# B&R Automation Studio project Kesim
Automation Studio 6.7.0.187; technology packages: mappCockpit 6.7.0, mappMotion 6.7.2, mappServices 6.7.1, mappView 6.7.0, OpcUaCs 6.7.0

## Configuration Config1

CPU X20CP1685, AutomationRuntime 6.7.6, Build 11.3.0, Vc 6.5.0

### Task classes (Cpu.sw)
```
Cyclic#4:
  Kesim <- SourceCode.Kesim.prg
  CncCtrl <- SourceCode.CncCtrl.prg
Libraries: MpBase, runtime, AsZip, FileIO, aLibFile, AsBrStr, standard, astime, sys_lib, McBase, MpAxis, McAcpAx, McPathGen, McAcpTrak, McAxGroup, McAxis, McProgInt, MpRecipe, MpUserX, MpCnc, MpFile, MpPackML, MpAlarmX, CoTrace, MpServer, CMS_CT
```

### Hardware
```
8EI8X8HWT10.xxxx-1 : 8EI8X8HWT10.xxxx-1 v2.4.0.0 (NodeNumber=1)  [PLK1 -> X20CP1685.IF3 [Cable Type=PowerlinkCable, Length=10, Version=1.0.0.3]]
  DriveConfiguration/Encoder/EncoderX41:
    InterfaceType = EnDat
  DriveConfiguration/Encoder/EncoderX42:
    InterfaceType = EnDat
  DriveConfiguration/Encoder/EncoderX43:
    InterfaceType = EnDat
  DriveConfiguration/Channel[1]/RealAxis:
    AxisReference = gMpLink_AxisQX
  DriveConfiguration/Channel[1]/RealAxis/Homing:
    RestorePositionVariable = 
  DriveConfiguration/Channel[2]/RealAxis:
    AxisReference = gMpLink_AxisQY
  DriveConfiguration/Channel[2]/RealAxis/Homing:
    RestorePositionVariable = 
  DriveConfiguration/Channel[3]/RealAxis:
    AxisReference = gMpLink_AxisQC
  DriveConfiguration/Channel[3]/RealAxis/Homing:
    RestorePositionVariable = 
X20CP1685 : X20CP1685 v1.9.0.0
  Connector IF2:
    ActivateDevice = 1
    Mode = Manual
    InternetAddress = 192.168.5.10
    SubnetMask = 255.255.255.0
  ConfigurationID = Kesim_Config1
  Simulation = 1
  MotionLoggerSize = 2048000
  FileDevice1
  FileDeviceName1 = USER
  FileDevicePath1 = USER_PATH
```

### AxesGroup.axesgroup - X20CP1685/mappMotion/3AxesCNCXYC/AxesGroup.axesgroup
```
Element gMpLink_CncXYZ (Type=axesgroup)
  Type = PathGenAxesGroup
    PhysicalAxes:
      JointAxes:
        JointAxis[1]:
          Name = QX
          AxisRef = gMpLink_AxisQX
        JointAxis[2]:
          Name = QY
          AxisRef = gMpLink_AxisQY
        JointAxis[3]:
          Name = QZ
          AxisRef = gMpLink_AxisQC
    MechanicalSystem:
      MechSysRef = MechSys_3AxCNCXYZ
    AxesGroupFeatures:
      FeatureRef[1] = Feature_Programs
      FeatureRef[2] = Feature_Jogging
  Alarms = None
```

### CNCAxisCfg.axis - X20CP1685/mappMotion/3AxesCNCXYC/CNCAxisCfg.axis
```
Element gMpLink_AxisQX (Type=axis)
  BaseType = LinearBounded
  MovementLimits = Internal
    Position:
      LowerLimit = -25000.0
      UpperLimit = 25000.0
    Velocity:
      Velocity = 500000.0
    Acceleration:
      Acceleration = 500000.0
    Deceleration:
      Deceleration = 500000.0
  Alarms = None
Element gMpLink_AxisQY (Type=axis)
  BaseType = LinearBounded
  MovementLimits = Internal
    Position:
      LowerLimit = -25000.0
      UpperLimit = 25000.0
    Velocity:
      Velocity = 500000.0
    Acceleration:
      Acceleration = 500000.0
    Deceleration:
      Deceleration = 500000.0
  Alarms = None
Element gMpLink_AxisQC (Type=axis)
  BaseType = RotaryBounded
  MovementLimits = Internal
    Position:
      LowerLimit = -25000.0
      UpperLimit = 25000.0
    Velocity:
      Velocity = 500000.0
    Acceleration:
      Acceleration = 500000.0
    Deceleration:
      Deceleration = 500000.0
  Alarms = None
```

### GroupFeat.axesgroupfeature - X20CP1685/mappMotion/3AxesCNCXYC/GroupFeat.axesgroupfeature
```
Element Feature_Programs (Type=axesgroupfeature)
  Type = Program
    Location = User
      UserLocation[1]:
        FileDevice = DEV_CNC
Element Feature_Jogging (Type=axesgroupfeature)
  Type = Jogging
```

### MotionCfg.mappmotioncfg - X20CP1685/mappMotion/MotionCfg.mappmotioncfg
```
Element MappMotionConfiguration (Type=mappmotioncfg)
  SharedAlarms:
    Axis = MpAlarmX
    ACOPOSmultiAuxiliarySupplyModule = MpAlarmX
    ACOPOSmultiPowerSupplyModule = MpAlarmX
    AxesGroup = MpAlarmX
    Assembly = MpAlarmX
    Segment = MpAlarmX
    Sector = MpAlarmX
    Shuttle = MpAlarmX
    CamOperations = MpAlarmX
  Diagnostics:
    Snapshot = NotUsed
```

### AlmXCore.mpalarmxcore - X20CP1685/mappServices/AlarmX/AlmXCore.mpalarmxcore
```
Element gMpLink_AlarmXCore (Type=mpalarmxcore)
  mapp.Gen:
    Enable = TRUE
    EnableCockpit = TRUE
    TaskClass = 1
    Parent
  mapp.AlarmX.Core:
    Mapping:
      [0]:
        Alarm = [0]
        Action = Reaction
          Name = Category0_Abort
      [1]:
        Alarm = [1]
        Action = Reaction
          Name = Category1_Stop
      [2]:
        Alarm = [2]
        Action = Reaction
          Name = Category2_Pause
      [3]:
        Alarm = [3]
        Action = Reaction
          Name = Category3_Info
  mapp.AlarmX.List:
    [0]:
      List = gMpLink_AlarmXList_Abort
      Offset = 0
    [1]:
      List = gMpLink_AlarmXList_Stop
      Offset = 0
    [2]:
      List = gMpLink_AlarmXList_Info
      Offset = 0
  mapp.AlarmX.Create = Disabled
  mapp.AlarmX.Core.Retain:
    Memory = 0
  mapp.AlarmX.Core.Categories:
    [0]:
      List = gMpLink_AlarmXCategory
```

- AlmXLAbort.mpalarmxlist (1706109 bytes, not shown)

### RecipeXml.mprecipexml - X20CP1685/mappServices/Recipe/RecipeXml.mprecipexml
```
Element gMpLink_RecipeXml_Product (Type=mprecipexml)
  mapp.Gen:
    Enable = TRUE
    EnableCockpit = TRUE
    TaskClass = 4
    Audit = TRUE
    Parent
  mapp.Recipe.Xml:
    AutoSave = Standard
    Encryption = FALSE
    PassPhrase
    AutoExtension = TRUE
    Signature = Disabled
  Alarms = MpAlarmX
    mapp.AlarmX.Core.Configuration:
      [0]:
        Name = SaveFailed
        Message = {$BR/mapp/MpRecipeXml/Alarms/SaveFailed}
        Code = 0
        Severity = 1
        Behavior = EdgeAlarm
          AutoReset = TRUE
          Acknowledge = 1
          Confirm = 0
          MultipleInstances = TRUE
          ReactionWhilePending = TRUE
          Async = FALSE
          Recording:
            InactiveToActive = TRUE
            ActiveToInactive = FALSE
            UnacknowledgedToAcknowledged = TRUE
            UnconfirmedToConfirmed = TRUE
        Disable = FALSE
        AdditionalInformation1
        AdditionalInformation2
      [1]:
        Name = SaveFailedPartial
        Message = {$BR/mapp/MpRecipeXml/Alarms/SaveFailedPartial}
        Code = 0
        Severity = 1
        Behavior = EdgeAlarm
          AutoReset = TRUE
          Acknowledge = 1
          Confirm = 0
          MultipleInstances = TRUE
          ReactionWhilePending = TRUE
          Async = FALSE
          Recording:
            InactiveToActive = TRUE
            ActiveToInactive = FALSE
            UnacknowledgedToAcknowledged = TRUE
            UnconfirmedToConfirmed = TRUE
        Disable = FALSE
        AdditionalInformation1
        AdditionalInformation2
      [2]:
        Name = LoadFailed
        Message = {$BR/mapp/MpRecipeXml/Alarms/LoadFailed}
        Code = 0
        Severity = 1
        Behavior = EdgeAlarm
          AutoReset = TRUE
          Acknowledge = 1
          Confirm = 0
          MultipleInstances = TRUE
          ReactionWhilePending = TRUE
          Async = FALSE
          Recording:
            InactiveToActive = TRUE
            ActiveToInactive = FALSE
            UnacknowledgedToAcknowledged = TRUE
            UnconfirmedToConfirmed = TRUE
        Disable = FALSE
        AdditionalInformation1
        AdditionalInformation2
      [3]:
        Name = LoadFailedPartial
        Message = {$BR/mapp/MpRecipeXml/Alarms/LoadFailedPartial}
        Code = 0
        Severity = 1
        Behavior = EdgeAlarm
          AutoReset = TRUE
          Acknowledge = 1
          Confirm = 0
          MultipleInstances = TRUE
          ReactionWhilePending = TRUE
          Async = FALSE
          Recording:
            InactiveToActive = TRUE
            ActiveToInactive = FALSE
            UnacknowledgedToAcknowledged = TRUE
            UnconfirmedToConfirmed = TRUE
        Disable = FALSE
        AdditionalInformation1
        AdditionalInformation2
Element gMpLink_RecipeXml_Machine (Type=mprecipexml)
  mapp.Gen:
    Enable = TRUE
    EnableCockpit = TRUE
    TaskClass = 4
    Audit = TRUE
    Parent
  mapp.Recipe.Xml:
    AutoSave = Standard
    Encryption = FALSE
    PassPhrase
    AutoExtension = TRUE
    Signature = Disabled
  Alarms = MpAlarmX
    mapp.AlarmX.Core.Configuration:
      [0]:
        Name = SaveFailed
        Message = {$BR/mapp/MpRecipeXml/Alarms/SaveFailed}
        Code = 0
        Severity = 1
        Behavior = EdgeAlarm
          AutoReset = TRUE
          Acknowledge = 1
          Confirm = 0
          MultipleInstances = TRUE
          ReactionWhilePending = TRUE
          Async = FALSE
          Recording:
            InactiveToActive = TRUE
            ActiveToInactive = FALSE
            UnacknowledgedToAcknowledged = TRUE
            UnconfirmedToConfirmed = TRUE
        Disable = FALSE
        AdditionalInformation1
        AdditionalInformation2
      [1]:
        Name = SaveFailedPartial
        Message = {$BR/mapp/MpRecipeXml/Alarms/SaveFailedPartial}
        Code = 0
        Severity = 1
        Behavior = EdgeAlarm
          AutoReset = TRUE
          Acknowledge = 1
          Confirm = 0
          MultipleInstances = TRUE
          ReactionWhilePending = TRUE
          Async = FALSE
          Recording:
            InactiveToActive = TRUE
            ActiveToInactive = FALSE
            UnacknowledgedToAcknowledged = TRUE
            UnconfirmedToConfirmed = TRUE
        Disable = FALSE
        AdditionalInformation1
        AdditionalInformation2
      [2]:
        Name = LoadFailed
        Message = {$BR/mapp/MpRecipeXml/Alarms/LoadFailed}
        Code = 0
        Severity = 1
        Behavior = EdgeAlarm
          AutoReset = TRUE
          Acknowledge = 1
          Confirm = 0
          MultipleInstances = TRUE
          ReactionWhilePending = TRUE
          Async = FALSE
          Recording:
            InactiveToActive = TRUE
            ActiveToInactive = FALSE
            UnacknowledgedToAcknowledged = TRUE
            UnconfirmedToConfirmed = TRUE
        Disable = FALSE
        AdditionalInformation1
        AdditionalInformation2
      [3]:
        Name = LoadFailedPartial
        Message = {$BR/mapp/MpRecipeXml/Alarms/LoadFailedPartial}
        Code = 0
        Severity = 1
        Behavior = EdgeAlarm
          AutoReset = TRUE
          Acknowledge = 1
          Confirm = 0
          MultipleInstances = TRUE
          ReactionWhilePending = TRUE
          Async = FALSE
          Recording:
            InactiveToActive = TRUE
            ActiveToInactive = FALSE
            UnacknowledgedToAcknowledged = TRUE
            UnconfirmedToConfirmed = TRUE
        Disable = FALSE
        AdditionalInformation1
        AdditionalInformation2
```

### UsrX.mpuserx - X20CP1685/mappServices/UserX/UsrX.mpuserx
```
Element UserMgmtX (Type=mpuserx)
  mapp.Gen:
    Audit = TRUE
  UserMgmtSystem:
    UserMgmtSystemType = 0
  ServerSettings:
    Server = ADServer
      Timeout = 10
      Mapping:
        TableName
      DisplayName = Username
      AdditionalUserData:
        [0] = mail
        [1] = telephoneNumber
  PasswordPolicy:
    PasswordMaxAge = 0
    PasswordExpirationNotification = 0
    PasswordHistory = 0
    PasswordChangeReq = FALSE
    PasswordCase = FALSE
    PasswordAlpha = FALSE
    PasswordSpecial = FALSE
    PasswordLength = 2
  UserAccount:
    InvalidPasswordAttempts = 5
    UserExpirationTime = 0
    AutoLogoutTime = 3600
    UserNameLength = 1
    NoDelete = FALSE
    AdminUnlockTime = 0
    EditSameLevel = 1
  ImportExport:
    ImportUser = 2
    ImportRole = 2
    ImportUnchecked = FALSE
  Roles:
    DefRole#1:
      id = AdministratorBR
      level = 100
      admin = TRUE
    DefRole#2:
      id = AdministratorCU
      level = 90
      admin = TRUE
    DefRole#3:
      id = Supervisor
      level = 80
      admin = TRUE
    DefRole#4:
      id = Operator
      level = 70
      admin = TRUE
```

## Configuration FCL

CPU X20CP1685, AutomationRuntime 6.7.6, Build 11.3.0

### Hardware
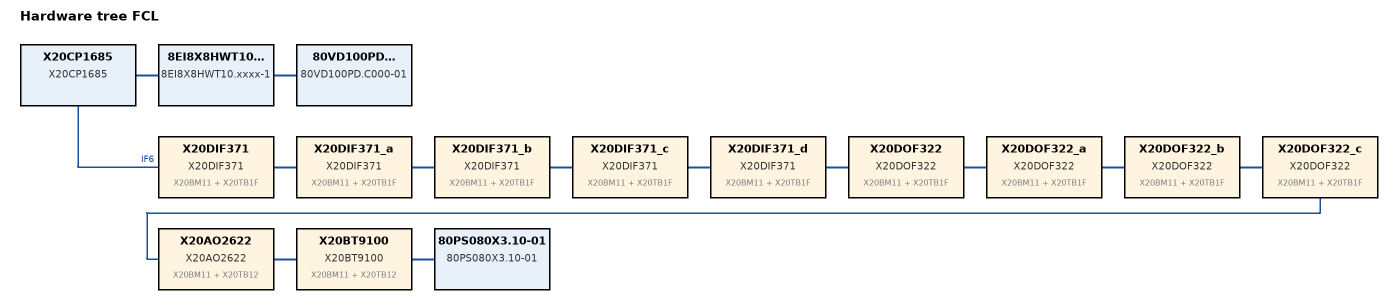
```
80PS080X3.10-01 : 80PS080X3.10-01 v1.7.0.0  [X2X1 -> X20BT9100.X2X1 [Cable Type=X2XCable, Length=10, Version=1.0.0.3]]
80VD100PD.C000-01 : 80VD100PD.C000-01 v2.5.1.0 (NodeNumber=2)  [PLK1 -> 8EI8X8HWT10.xxxx-1.PLK2 [Cable Type=PowerlinkCable, Length=10, Version=1.0.0.3]]
  EnableDNA = on
8EI8X8HWT10.xxxx-1 : 8EI8X8HWT10.xxxx-1 v2.4.0.0 (NodeNumber=1)  [PLK1 -> X20CP1685.IF3 [Cable Type=PowerlinkCable, Length=10, Version=1.0.0.3]; PLK2 -> 80VD100PD.C000-01.PLK1 [Cable Type=PowerlinkCable, Length=10, Version=1.0.0.3]]
  EnableDNA = on
X20AO2622 : X20AO2622 v1.5.0.0  [SS1 -> X20TB12.SS; SL -> X20BM11_i.SL1]
X20BM11 : X20BM11 v1.1.0.0  [X2X1 -> X20CP1685.IF6]
X20BM11_a : X20BM11 v1.1.0.0  [X2X1 -> X20BM11.X2X2]
X20BM11_b : X20BM11 v1.1.0.0  [X2X1 -> X20BM11_a.X2X2]
X20BM11_c : X20BM11 v1.1.0.0  [X2X1 -> X20BM11_b.X2X2]
X20BM11_d : X20BM11 v1.1.0.0  [X2X1 -> X20BM11_c.X2X2]
X20BM11_e : X20BM11 v1.1.0.0  [X2X1 -> X20BM11_d.X2X2]
X20BM11_f : X20BM11 v1.1.0.0  [X2X1 -> X20BM11_e.X2X2]
X20BM11_g : X20BM11 v1.1.0.0  [X2X1 -> X20BM11_f.X2X2]
X20BM11_h : X20BM11 v1.1.0.0  [X2X1 -> X20BM11_g.X2X2]
X20BM11_i : X20BM11 v1.1.0.0  [X2X1 -> X20BM11_h.X2X2]
X20BM11_j : X20BM11 v1.1.0.0  [X2X1 -> X20BM11_i.X2X2]
X20BT9100 : X20BT9100 v1.4.0.0  [SS1 -> X20TB12_a.SS; SL -> X20BM11_j.SL1]
X20CP1685 : X20CP1685 v1.9.0.0
  Connector IF2:
    ActivateDevice = 1
  ConfigurationID = Kesim_Config1
  Simulation = 1
  FileDevice1
  FileDeviceName1 = USER
  FileDevicePath1 = USER_PATH
X20DIF371 : X20DIF371 v1.4.1.0  [SS1 -> X20TB1F.SS; SL -> X20BM11.SL1]
X20DIF371_a : X20DIF371 v1.4.1.0  [SS1 -> X20TB1F_a.SS; SL -> X20BM11_a.SL1]
X20DIF371_b : X20DIF371 v1.4.1.0  [SS1 -> X20TB1F_b.SS; SL -> X20BM11_b.SL1]
X20DIF371_c : X20DIF371 v1.4.1.0  [SS1 -> X20TB1F_c.SS; SL -> X20BM11_c.SL1]
X20DIF371_d : X20DIF371 v1.4.1.0  [SS1 -> X20TB1F_d.SS; SL -> X20BM11_d.SL1]
X20DOF322 : X20DOF322 v1.5.2.0  [SS1 -> X20TB1F_e.SS; SL -> X20BM11_e.SL1]
X20DOF322_a : X20DOF322 v1.5.2.0  [SS1 -> X20TB1F_f.SS; SL -> X20BM11_f.SL1]
X20DOF322_b : X20DOF322 v1.5.2.0  [SS1 -> X20TB1F_g.SS; SL -> X20BM11_g.SL1]
X20DOF322_c : X20DOF322 v1.5.2.0  [SS1 -> X20TB1F_h.SS; SL -> X20BM11_h.SL1]
X20TB12 : X20TB12 v1.0.0.0
X20TB12_a : X20TB12 v1.0.0.0
X20TB1F : X20TB1F v1.0.0.0
X20TB1F_a : X20TB1F v1.0.0.0
X20TB1F_b : X20TB1F v1.0.0.0
X20TB1F_c : X20TB1F v1.0.0.0
X20TB1F_d : X20TB1F v1.0.0.0
X20TB1F_e : X20TB1F v1.0.0.0
X20TB1F_f : X20TB1F v1.0.0.0
X20TB1F_g : X20TB1F v1.0.0.0
X20TB1F_h : X20TB1F v1.0.0.0
```

## Configuration OCKM

### Hardware
```
X20CP1685 : X20CP1685 v1.9.0.0
  Connector IF2:
    ActivateDevice = 1
  ConfigurationID = Kesim_Config1
  Simulation = 1
  FileDevice1
  FileDeviceName1 = USER
  FileDevicePath1 = USER_PATH
```

## Configuration Office

CPU X20CP1685, AutomationRuntime 6.7.6, Build 11.3.0

### Task classes (Cpu.sw)
```
Cyclic#1:
  CncCtrl <- Source.CncCtrl.prg
Cyclic#4:
  AlarmX <- Source.Infastructure.AlarmX.prg
  UserXMgr <- Source.Infastructure.UserXMgr.prg
DataObjects: McAcpSys
NcDataObjects: McDriveLog
Binaries: TCLang, FWRules, mvLoader, TCData, udbdef, ArSvcReg, McAcpSim, McAcpDrv, McMechSys, iomap, asfw, Role, ashwd, sysconf, TC, BRRole, arconfig, User, ashwac, UaCsConfig, mCoWebSc, AxesGroup, SyncModule, CNCAxisCfg, MotionCfg, GroupFeat, Settings, SyncUnit, MechSystem, Hierarchy, mvConfig, AlmXCore, UsrX, AlmXHist, AlmXList, AlmXCateg, UsrXLogin, RecipeXml
Libraries: ArSsl, DataObj, UaCoal, AsHW, ArCert, ArUser, UaCoalPrv, AsETH, powerlnk, AsArProf, brsystem, AsMem, AsIO, AsEPL, operator, runtime, AsIecCon, astime, aLibFile, FileIO, AsBrStr, standard, sys_lib, AsZip, McBase, MpBase, MpAxis, McAcpAx, McPathGen, McAcpTrak, McAxGroup, McAxis, McProgInt, MpCnc, CoTrace, MpRecipe, MpUserX, MpFile, MpPackML, MpAlarmX, MpServer, CMS_CT
```

### Hardware
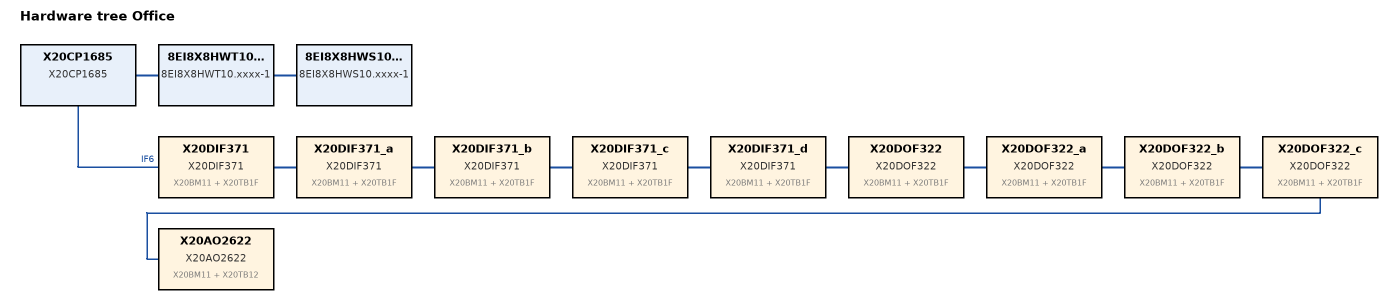
```
8EI8X8HWS10.xxxx-1 : 8EI8X8HWS10.xxxx-1 v2.4.0.0 (NodeNumber=2)  [PLK1 -> 8EI8X8HWT10.xxxx-1.PLK2 [Cable Type=PowerlinkCable, Length=10, Version=1.0.0.3]]
8EI8X8HWT10.xxxx-1 : 8EI8X8HWT10.xxxx-1 v2.4.0.0 (NodeNumber=1)  [PLK1 -> X20CP1685.IF3 [Cable Type=PowerlinkCable, Length=10, Version=1.0.0.3]; PLK2 -> 8EI8X8HWS10.xxxx-1.PLK1 [Cable Type=PowerlinkCable, Length=10, Version=1.0.0.3]]
  DriveConfiguration/Module:
    McAcoposTypeID = AcoposP3TConfig
    ActivateACOPOSSimulationOnPLC = 0
    PowerSupply = AC
  DriveConfiguration/Encoder/EncoderX41:
    InterfaceType = EnDat
  DriveConfiguration/Encoder/EncoderX42:
    InterfaceType = EnDat
  DriveConfiguration/Encoder/EncoderX43:
    InterfaceType = EnDat
  DriveConfiguration/Channel[1]/RealAxis:
    AxisReference = gMpLink_AxisQX
    MechanicalElementsIsInvisible = 0
  DriveConfiguration/Channel[1]/RealAxis/MechanicalElements/Gearbox:
    InputIsReadOnly = 0
    Input = 1
    OutputIsReadOnly = 0
    Output = 1
  DriveConfiguration/Channel[1]/RealAxis/MechanicalElements/RotaryToLinearTransformation:
    ReferenceDistanceIsReadOnly = 0
    ReferenceDistance = 1
  DriveConfiguration/Channel[1]/RealAxis:
    EncoderLink = OneEncoder
  DriveConfiguration/Channel[1]/RealAxis/Controller:
    ModeIsReadOnly = 0
    Mode = PositionController
  DriveConfiguration/Channel[1]/RealAxis/Homing:
    ModeIsReadOnly = 0
    Mode = Direct
    RestorePositionVariable = 
  DriveConfiguration/Channel[1]/RealAxis/StopReaction:
    QuickstopIsReadOnly = 0
    Quickstop = DecelerationLimit
    DriveErrorIsReadOnly = 0
    DriveError = DecelerationLimit
  DriveConfiguration/Channel[1]/RealAxis/MovementErrorLimits:
    PositionError = 10.0
    VelocityErrorMonitoring = Automatic1
  DriveConfiguration/Channel[1]/RealAxis:
    JerkFilterIsReadOnly = 0
    JerkFilter = NotUsed
    ZeroVibrationFilter = NotUsed
  DriveConfiguration/Channel[1]/RealAxis/DigitalInputs/HomingSwitch:
    SourceIsReadOnly = 0
    Source = NotUsed
    Level = High
  DriveConfiguration/Channel[1]/RealAxis/DigitalInputs/PositiveLimitSwitch:
    SourceIsReadOnly = 0
    Source = NotUsed
    Level = High
  DriveConfiguration/Channel[1]/RealAxis/DigitalInputs/NegativeLimitSwitch:
    SourceIsReadOnly = 0
    Source = NotUsed
    Level = High
  DriveConfiguration/Channel[1]/RealAxis/DigitalInputs/Trigger1:
    Source = X8Trigger1
    Level = High
  DriveConfiguration/Channel[1]/RealAxis/DigitalInputs/Trigger2:
    Source = X8Trigger2
    Level = High
  DriveConfiguration/Channel[1]/RealAxis/DigitalInputs/Quickstop:
    Input = Trigger2
  DriveConfiguration/Channel[1]/RealAxis/Simulation:
    SimulationModeOnPLC = SetValueGeneration
    SimulationModeOnACOPOS = NotUsed
  DriveConfiguration/Channel[1]:
    VirtualAxis = NotUsed
    ExternalEncoderAxis = NotUsed
  DriveConfiguration/Channel[2]/RealAxis:
    AxisReference = gMpLink_AxisQY
    MechanicalElementsIsInvisible = 0
  DriveConfiguration/Channel[2]/RealAxis/MechanicalElements/Gearbox:
    InputIsReadOnly = 0
    Input = 1
    OutputIsReadOnly = 0
    Output = 1
  DriveConfiguration/Channel[2]/RealAxis/MechanicalElements/RotaryToLinearTransformation:
    ReferenceDistanceIsReadOnly = 0
    ReferenceDistance = 1
  DriveConfiguration/Channel[2]/RealAxis:
    EncoderLink = OneEncoder
  DriveConfiguration/Channel[2]/RealAxis/Controller:
    ModeIsReadOnly = 0
    Mode = PositionController
  DriveConfiguration/Channel[2]/RealAxis/Homing:
    ModeIsReadOnly = 0
    Mode = Direct
    RestorePositionVariable = 
  DriveConfiguration/Channel[2]/RealAxis/StopReaction:
    QuickstopIsReadOnly = 0
    Quickstop = DecelerationLimit
    DriveErrorIsReadOnly = 0
    DriveError = DecelerationLimit
  DriveConfiguration/Channel[2]/RealAxis/MovementErrorLimits:
    PositionError = 10.0
    VelocityErrorMonitoring = Automatic1
  DriveConfiguration/Channel[2]/RealAxis:
    JerkFilterIsReadOnly = 0
    JerkFilter = NotUsed
    ZeroVibrationFilter = NotUsed
  DriveConfiguration/Channel[2]/RealAxis/DigitalInputs/HomingSwitch:
    SourceIsReadOnly = 0
    Source = NotUsed
    Level = High
  DriveConfiguration/Channel[2]/RealAxis/DigitalInputs/PositiveLimitSwitch:
    SourceIsReadOnly = 0
    Source = NotUsed
    Level = High
  DriveConfiguration/Channel[2]/RealAxis/DigitalInputs/NegativeLimitSwitch:
    SourceIsReadOnly = 0
    Source = NotUsed
    Level = High
  DriveConfiguration/Channel[2]/RealAxis/DigitalInputs/Trigger1:
    Source = X8Trigger1
    Level = High
  DriveConfiguration/Channel[2]/RealAxis/DigitalInputs/Trigger2:
    Source = X8Trigger2
    Level = High
  DriveConfiguration/Channel[2]/RealAxis/DigitalInputs/Quickstop:
    Input = Trigger2
  DriveConfiguration/Channel[2]/RealAxis/Simulation:
    SimulationModeOnPLC = SetValueGeneration
    SimulationModeOnACOPOS = NotUsed
  DriveConfiguration/Channel[2]:
    VirtualAxis = NotUsed
    ExternalEncoderAxis = NotUsed
  DriveConfiguration/Channel[3]/RealAxis:
    AxisReference = gMpLink_AxisQC
    MechanicalElementsIsInvisible = 0
  DriveConfiguration/Channel[3]/RealAxis/MechanicalElements/Gearbox:
    InputIsReadOnly = 0
    Input = 1
    OutputIsReadOnly = 0
    Output = 1
  DriveConfiguration/Channel[3]/RealAxis/MechanicalElements/RotaryToLinearTransformation:
    ReferenceDistanceIsReadOnly = 0
    ReferenceDistance = 1
  DriveConfiguration/Channel[3]/RealAxis:
    EncoderLink = OneEncoder
  DriveConfiguration/Channel[3]/RealAxis/Controller:
    ModeIsReadOnly = 0
    Mode = PositionController
  DriveConfiguration/Channel[3]/RealAxis/Homing:
    ModeIsReadOnly = 0
    Mode = Direct
    RestorePositionVariable = 
  DriveConfiguration/Channel[3]/RealAxis/StopReaction:
    QuickstopIsReadOnly = 0
    Quickstop = DecelerationLimit
    DriveErrorIsReadOnly = 0
    DriveError = DecelerationLimit
  DriveConfiguration/Channel[3]/RealAxis/MovementErrorLimits:
    PositionError = 10.0
    VelocityErrorMonitoring = Automatic1
  DriveConfiguration/Channel[3]/RealAxis:
    JerkFilterIsReadOnly = 0
    JerkFilter = NotUsed
    ZeroVibrationFilter = NotUsed
  DriveConfiguration/Channel[3]/RealAxis/DigitalInputs/HomingSwitch:
    SourceIsReadOnly = 0
    Source = NotUsed
    Level = High
  DriveConfiguration/Channel[3]/RealAxis/DigitalInputs/PositiveLimitSwitch:
    SourceIsReadOnly = 0
    Source = NotUsed
    Level = High
  DriveConfiguration/Channel[3]/RealAxis/DigitalInputs/NegativeLimitSwitch:
    SourceIsReadOnly = 0
    Source = NotUsed
    Level = High
  DriveConfiguration/Channel[3]/RealAxis/DigitalInputs/Trigger1:
    Source = X8Trigger1
    Level = High
  DriveConfiguration/Channel[3]/RealAxis/DigitalInputs/Trigger2:
    Source = X8Trigger2
    Level = High
  DriveConfiguration/Channel[3]/RealAxis/DigitalInputs/Quickstop:
    Input = Trigger2
  DriveConfiguration/Channel[3]/RealAxis/Simulation:
    SimulationModeOnPLC = SetValueGeneration
    SimulationModeOnACOPOS = NotUsed
  DriveConfiguration/Channel[3]:
    VirtualAxis = NotUsed
    ExternalEncoderAxis = NotUsed
X20AO2622 : X20AO2622 v1.5.0.0  [SS1 -> X20TB12.SS; SL -> X20BM11_i.SL1]
X20BM11 : X20BM11 v1.1.0.0  [X2X1 -> X20CP1685.IF6]
X20BM11_a : X20BM11 v1.1.0.0  [X2X1 -> X20BM11.X2X2]
X20BM11_b : X20BM11 v1.1.0.0  [X2X1 -> X20BM11_a.X2X2]
X20BM11_c : X20BM11 v1.1.0.0  [X2X1 -> X20BM11_b.X2X2]
X20BM11_d : X20BM11 v1.1.0.0  [X2X1 -> X20BM11_c.X2X2]
X20BM11_e : X20BM11 v1.1.0.0  [X2X1 -> X20BM11_d.X2X2]
X20BM11_f : X20BM11 v1.1.0.0  [X2X1 -> X20BM11_e.X2X2]
X20BM11_g : X20BM11 v1.1.0.0  [X2X1 -> X20BM11_f.X2X2]
X20BM11_h : X20BM11 v1.1.0.0  [X2X1 -> X20BM11_g.X2X2]
X20BM11_i : X20BM11 v1.1.0.0  [X2X1 -> X20BM11_h.X2X2]
X20CP1685 : X20CP1685 v1.9.0.0
  Connector IF2:
    ActivateDevice = 1
    ActivateSnmp = 2
  ConfigurationID = Cutting Table
  Simulation = 1
  MotionLoggerSize = 2048000
  EnableDebugger = 1
  TimerDeviceType = EPLX2X
  TimerDevice = X20CP1685.IF3
  TaskClassIdleTime = 2000
  Cyclic1Tolerance = 0
  FileDevice1
  FileDeviceName1 = USER
  FileDevicePath1 = USER_PATH
  ActivateFtpServer = 1
  ActivateWebServer = 1
  WebServerProtocol = 3
  ActivateSdm = 1
X20DIF371 : X20DIF371 v1.4.1.0  [SS1 -> X20TB1F.SS; SL -> X20BM11.SL1]
X20DIF371_a : X20DIF371 v1.4.1.0  [SS1 -> X20TB1F_a.SS; SL -> X20BM11_a.SL1]
X20DIF371_b : X20DIF371 v1.4.1.0  [SS1 -> X20TB1F_b.SS; SL -> X20BM11_b.SL1]
X20DIF371_c : X20DIF371 v1.4.1.0  [SS1 -> X20TB1F_c.SS; SL -> X20BM11_c.SL1]
X20DIF371_d : X20DIF371 v1.4.1.0  [SS1 -> X20TB1F_d.SS; SL -> X20BM11_d.SL1]
X20DOF322 : X20DOF322 v1.5.2.0  [SS1 -> X20TB1F_e.SS; SL -> X20BM11_e.SL1]
X20DOF322_a : X20DOF322 v1.5.2.0  [SS1 -> X20TB1F_f.SS; SL -> X20BM11_f.SL1]
X20DOF322_b : X20DOF322 v1.5.2.0  [SS1 -> X20TB1F_g.SS; SL -> X20BM11_g.SL1]
X20DOF322_c : X20DOF322 v1.5.2.0  [SS1 -> X20TB1F_h.SS; SL -> X20BM11_h.SL1]
X20TB12 : X20TB12 v1.0.0.0
X20TB1F : X20TB1F v1.0.0.0
X20TB1F_a : X20TB1F v1.0.0.0
X20TB1F_b : X20TB1F v1.0.0.0
X20TB1F_c : X20TB1F v1.0.0.0
X20TB1F_d : X20TB1F v1.0.0.0
X20TB1F_e : X20TB1F v1.0.0.0
X20TB1F_f : X20TB1F v1.0.0.0
X20TB1F_g : X20TB1F v1.0.0.0
X20TB1F_h : X20TB1F v1.0.0.0
```

### IoMap.iom - X20CP1685/IoMap.iom
```iecst
VAR_CONFIG
	::Kesim:fbCuttingTransfer_0.inEnable AT %IX."X20DIF371".DigitalInput01;
END_VAR
```

### PvMap.vvm - X20CP1685/PvMap.vvm
```iecst
VAR_CONFIG
	Cyclic#1.::ForceIO:slotIndex AT %Q.Cyclic#1.::gHMI.IO_Control.SelectedSlot; (*Insert your comment here...*)
	Cyclic#1.::ForceIO:GetSignalStr_0.eTypeSignal AT %Q.Cyclic#1.::gHMI.IO_Control.TypeOfIO; (*Insert your comment here...*)
END_VAR
```

### AxesGroup.axesgroup - X20CP1685/mappMotion/3AxesCNCXYC/AxesGroup.axesgroup
```
Element gMpLink_CncXYZ (Type=axesgroup)
  Type = PathGenAxesGroup
    PhysicalAxes:
      JointAxes:
        JointAxis[1]:
          Name = QX
          AxisRef = gMpLink_AxisQX
        JointAxis[2]:
          Name = QY
          AxisRef = gMpLink_AxisQY
        JointAxis[3]:
          Name = QC
          AxisRef = gMpLink_AxisQC
    MechanicalSystem:
      MechSysRef = MechSys_3AxCNCXYZ
    AxesGroupFeatures:
      FeatureRef[1] = Feature_Programs
      FeatureRef[2] = Feature_Jogging
```

### CNCAxisCfg.axis - X20CP1685/mappMotion/3AxesCNCXYC/CNCAxisCfg.axis
```
Element gMpLink_AxisQX (Type=axis)
  BaseType = LinearBounded
  MovementLimits = Internal
    Position:
      LowerLimit = -25000.0
      UpperLimit = 25000.0
    Velocity:
      Velocity = 500000.0
    Acceleration:
      Acceleration = 500000.0
    Deceleration:
      Deceleration = 500000.0
  Alarms = None
Element gMpLink_AxisQY (Type=axis)
  BaseType = LinearBounded
  MovementLimits = Internal
    Position:
      LowerLimit = -25000.0
      UpperLimit = 25000.0
    Velocity:
      Velocity = 500000.0
    Acceleration:
      Acceleration = 500000.0
    Deceleration:
      Deceleration = 500000.0
  Alarms = None
Element gMpLink_AxisQC (Type=axis)
  BaseType = RotaryBounded
  MovementLimits = Internal
    Position:
      LowerLimit = -25000.0
      UpperLimit = 25000.0
    Velocity:
      Velocity = 500000.0
    Acceleration:
      Acceleration = 500000.0
    Deceleration:
      Deceleration = 500000.0
  Alarms = None
```

### AxesGroup.axesgroup - X20CP1685/mappMotion/3AxesCNCXYZ/AxesGroup.axesgroup
```
Element gMpLink_CncXYZ (Type=axesgroup)
  Type = PathGenAxesGroup
    PhysicalAxes:
      JointAxes:
        JointAxis[1]:
          Name = QX
          AxisRef = gMpLink_AxisQX
        JointAxis[2]:
          Name = QY
          AxisRef = gMpLink_AxisQY
        JointAxis[3]:
          Name = VQZ
          AxisRef = gMpLink_AxisVQZ
    MechanicalSystem:
      MechSysRef = MechSys_3AxCNCXYZ
    AxesGroupFeatures:
      FeatureRef[1] = Feature_Programs
      FeatureRef[2] = Feature_Jogging
```

### CNCAxisCfg.axis - X20CP1685/mappMotion/3AxesCNCXYZ/CNCAxisCfg.axis
```
Element gMpLink_AxisQX (Type=axis)
  BaseType = LinearBounded
  MovementLimits:
    Position:
      LowerLimit = -25000.0
      UpperLimit = 25000.0
    Velocity:
      Velocity = 500000.0
    Acceleration:
      Acceleration = 500000.0
    Deceleration:
      Deceleration = 500000.0
Element gMpLink_AxisQY (Type=axis)
  BaseType = LinearBounded
  MovementLimits:
    Position:
      LowerLimit = -25000.0
      UpperLimit = 25000.0
    Velocity:
      Velocity = 500000.0
    Acceleration:
      Acceleration = 500000.0
    Deceleration:
      Deceleration = 500000.0
Element gMpLink_AxisVQZ (Type=axis)
  BaseType = LinearBounded
  MovementLimits:
    Position:
      LowerLimit = -25000.0
      UpperLimit = 25000.0
    Velocity:
      Velocity = 500000.0
    Acceleration:
      Acceleration = 500000.0
    Deceleration:
      Deceleration = 500000.0
Element gMpLink_AxisB (Type=axis)
  BaseType = RotaryBounded
  MovementLimits:
    Position:
      LowerLimit = -25000.0
      UpperLimit = 25000.0
    Velocity:
      Velocity = 500000.0
    Acceleration:
      Acceleration = 500000.0
    Deceleration:
      Deceleration = 500000.0
Element gMpLink_AxisC (Type=axis)
  BaseType = RotaryBounded
  MovementLimits:
    Position:
      LowerLimit = -25000.0
      UpperLimit = 25000.0
    Velocity:
      Velocity = 500000.0
    Acceleration:
      Acceleration = 500000.0
    Deceleration:
      Deceleration = 500000.0
```

### MechSystem.mechanicalsystem - X20CP1685/mappMotion/3AxesCNCXYZ/MechSystem.mechanicalsystem
```
Element MechSys_3AxCNCXYZ (Type=mechanicalsystem)
  Type = 3AxesCNC
    Subtype:
      JointAxesPositionLimits:
        JointAxis[1]
        JointAxis[2]
        JointAxis[3]
```

### MotionCfg.mappmotioncfg - X20CP1685/mappMotion/MotionCfg.mappmotioncfg
```
Element MappMotionConfiguration (Type=mappmotioncfg)
  Processing:
    ProcessingTaskClass = 1
    ExplicitComputationOrder:
      Axis = NotUsed
  Logger:
    SelectiveLogging = NotUsed
  SharedAlarms:
    Axis = MpAlarmX
    ACOPOSmultiAuxiliarySupplyModule = MpAlarmX
    ACOPOSmultiPowerSupplyModule = MpAlarmX
    AxesGroup = MpAlarmX
    Assembly = MpAlarmX
    Segment = MpAlarmX
    Sector = MpAlarmX
    Shuttle = MpAlarmX
    CamOperations = MpAlarmX
  McAcpDrv:
    POWERLINKCyclesPerParID = 2
```

### Config_3.purevaxcfg - X20CP1685/mappMotion/PureVAxis/Config_3.purevaxcfg
```
Element PureVAxCfg_1 (Type=purevaxcfg)
  PureVAxis:
    AxisReference = gMpLink_AxisVQZ
```

### AlmXCateg.mpalarmxcategory - X20CP1685/mappServices/AlarmX/AlmXCateg.mpalarmxcategory
```
Element gMpLink_AlarmXCategory (Type=mpalarmxcategory)
  mapp.AlarmX.Categories:
    [0]:
      Name = Category0_Abort
      SourceProperty = Severity
        Severity = 0
    [1]:
      Name = Category1_Stop
      SourceProperty = Severity
        Severity = 1
    [2]:
      Name = Category2_Pause
      SourceProperty = Severity
        Severity = 2
    [3]:
      Name = Category3_Info
      SourceProperty = Severity
        Severity = 3
```

### AlmXHist.mpalarmxhistory - X20CP1685/mappServices/AlarmX/AlmXHist.mpalarmxhistory
```
Element gMpLink_AlarmXHistory (Type=mpalarmxhistory)
  mapp.Gen:
    Enable = TRUE
    EnableCockpit = TRUE
    Audit = TRUE
    Parent
  mapp.AlarmX.History:
    Export:
      TimeStampPattern = %Y-%m-%d %H:%M:%S:%L
      AutoExtension = TRUE
      ColumnSeparator = ,
    Memory = 0
      Size = 2048
      BufferSize = 10
      Interval = 60
    Scope = 0
```

### AlmXLInfo.mpalarmxlist - X20CP1685/mappServices/AlarmX/AlmXLInfo.mpalarmxlist
```
Element gMpLink_AlarmXList_Info (Type=mpalarmxlist)
  mapp.AlarmX.Core.Configuration:
    [0]:
      Name = Alert.0
      Message = {&TextSnippet.0}{$AlarmX/Alerts/Alert.0}
      Code = 0
      Severity = 3
      Behavior = DiscreteValueMonitoring
        Confirm = 0
        ReactionWhilePending = TRUE
        Recording:
          InactiveToActive = TRUE
          UnacknowledgedToAcknowledged = TRUE
          AcknowledgedToUnacknowledged = FALSE
          UnconfirmedToConfirmed = TRUE
          ConfirmedToUnconfirmed = FALSE
          Update = FALSE
        Monitoring:
          MonitoredPV = ::AlarmX:Loc.Status.Alerts.Single.Info[0]
          TriggerValues:
            [0] = 1
          Settings = 0
            Delay = 0.0
      Disable = FALSE
      InhibitPV
      AdditionalInformation1
      AdditionalInformation2
    [1]:
      Name = Alert.1
      Message = {&TextSnippet.1}{$AlarmX/Alerts/Alert.1}
      Code = 1
      Severity = 2
      Behavior = DiscreteValueMonitoring
        Confirm = 0
        ReactionWhilePending = TRUE
        Recording:
          InactiveToActive = TRUE
          UnacknowledgedToAcknowledged = TRUE
          AcknowledgedToUnacknowledged = FALSE
          UnconfirmedToConfirmed = TRUE
          ConfirmedToUnconfirmed = FALSE
          Update = FALSE
        Monitoring:
          MonitoredPV = ::AlarmX:Loc.Status.Alerts.Single.Stop[1]
          TriggerValues:
            [0] = 1
          Settings = 0
            Delay = 0.0
      Disable = FALSE
      InhibitPV
      AdditionalInformation1
      AdditionalInformation2
    [2]:
      Name = Alert.2
      Message = {&TextSnippet.2}{$AlarmX/Alerts/Alert.2}
      Code = 2
      Severity = 2
      Behavior = DiscreteValueMonitoring
        Confirm = 0
        ReactionWhilePending = TRUE
        Recording:
          InactiveToActive = TRUE
          UnacknowledgedToAcknowledged = TRUE
          AcknowledgedToUnacknowledged = FALSE
          UnconfirmedToConfirmed = TRUE
          ConfirmedToUnconfirmed = FALSE
          Update = FALSE
        Monitoring:
          MonitoredPV = ::AlarmX:Loc.Status.Alerts.Single.Stop[2]
          TriggerValues:
            [0] = 1
          Settings = 0
            Delay = 0.0
      Disable = FALSE
      InhibitPV
      AdditionalInformation1
      AdditionalInformation2
    [3]:
      Name = Alert.3
      Message = {&TextSnippet.3}{$AlarmX/Alerts/Alert.3}
      Code = 3
      Severity = 2
      Behavior = DiscreteValueMonitoring
        Confirm = 0
        ReactionWhilePending = TRUE
        Recording:
          InactiveToActive = TRUE
          UnacknowledgedToAcknowledged = TRUE
          AcknowledgedToUnacknowledged = FALSE
          UnconfirmedToConfirmed = TRUE
          ConfirmedToUnconfirmed = FALSE
          Update = FALSE
        Monitoring:
          MonitoredPV = ::AlarmX:Loc.Status.Alerts.Single.Stop[3]
          TriggerValues:
            [0] = 1
          Settings = 0
            Delay = 0.0
      Disable = FALSE
      InhibitPV
      AdditionalInformation1
      AdditionalInformation2
    [4]:
      Name = Alert.4
      Message = {&TextSnippet.4}{$AlarmX/Alerts/Alert.4}
      Code = 4
      Severity = 2
      Behavior = DiscreteValueMonitoring
        Confirm = 0
        ReactionWhilePending = TRUE
        Recording:
          InactiveToActive = TRUE
          UnacknowledgedToAcknowledged = TRUE
          AcknowledgedToUnacknowledged = FALSE
          UnconfirmedToConfirmed = TRUE
          ConfirmedToUnconfirmed = FALSE
          Update = FALSE
        Monitoring:
          MonitoredPV = ::AlarmX:Loc.Status.Alerts.Single.Stop[4]
          TriggerValues:
            [0] = 1
          Settings = 0
            Delay = 0.0
      Disable = FALSE
      InhibitPV
      AdditionalInformation1
      AdditionalInformation2
    [5]:
      Name = Alert.5
      Message = {$AlarmX/Alerts/Alert.5}
      Code = 5
      Severity = 2
      Behavior = DiscreteValueMonitoring
        Confirm = 0
        ReactionWhilePending = TRUE
        Recording:
          InactiveToActive = TRUE
          UnacknowledgedToAcknowledged = TRUE
          AcknowledgedToUnacknowledged = FALSE
          UnconfirmedToConfirmed = TRUE
          ConfirmedToUnconfirmed = FALSE
          Update = FALSE
        Monitoring:
          MonitoredPV = ::AlarmX:Loc.Status.Alerts.Single.Stop[5]
          TriggerValues:
            [0] = 1
          Settings = 0
            Delay = 0.0
      Disable = FALSE
      InhibitPV
      AdditionalInformation1
      AdditionalInformation2
    [6]:
      Name = Alert.6
      Message = {$AlarmX/Alerts/Alert.6}
      Code = 6
      Severity = 2
      Behavior = DiscreteValueMonitoring
        Confirm = 0
        ReactionWhilePending = TRUE
        Recording:
          InactiveToActive = TRUE
          UnacknowledgedToAcknowledged = TRUE
          AcknowledgedToUnacknowledged = FALSE
          UnconfirmedToConfirmed = TRUE
          ConfirmedToUnconfirmed = FALSE
          Update = FALSE
        Monitoring:
          MonitoredPV = ::AlarmX:Loc.Status.Alerts.Single.Stop[6]
          TriggerValues:
            [0] = 1
          Settings = 0
            Delay = 0.0
      Disable = FALSE
      InhibitPV
      AdditionalInformation1
      AdditionalInformation2
    [7]:
      Name = Alert.7
      Message = {$AlarmX/Alerts/Alert.7}
      Code = 7
      Severity = 2
      Behavior = DiscreteValueMonitoring
        Confirm = 0
        ReactionWhilePending = TRUE
        Recording:
          InactiveToActive = TRUE
          UnacknowledgedToAcknowledged = TRUE
          AcknowledgedToUnacknowledged = FALSE
          UnconfirmedToConfirmed = TRUE
          ConfirmedToUnconfirmed = FALSE
          Update = FALSE
        Monitoring:
          MonitoredPV = ::AlarmX:Loc.Status.Alerts.Single.Stop[7]
          TriggerValues:
            [0] = 1
          Settings = 0
            Delay = 0.0
      Disable = FALSE
      InhibitPV
      AdditionalInformation1
      AdditionalInformation2
    [8]:
      Name = Alert.8
      Message = {$AlarmX/Alerts/Alert.8}
      Code = 8
      Severity = 2
      Behavior = DiscreteValueMonitoring
        Confirm = 0
        ReactionWhilePending = TRUE
        Recording:
          InactiveToActive = TRUE
          UnacknowledgedToAcknowledged = TRUE
          AcknowledgedToUnacknowledged = FALSE
          UnconfirmedToConfirmed = TRUE
          ConfirmedToUnconfirmed = FALSE
          Update = FALSE
        Monitoring:
          MonitoredPV = ::AlarmX:Loc.Status.Alerts.Single.Stop[8]
          TriggerValues:
            [0] = 1
          Settings = 0
            Delay = 0.0
      Disable = FALSE
      InhibitPV
      AdditionalInformation1
      AdditionalInformation2
    [9]:
      Name = Alert.9
      Message = {$AlarmX/Alerts/Alert.9}
      Code = 9
      Severity = 2
      Behavior = DiscreteValueMonitoring
        Confirm = 0
        ReactionWhilePending = TRUE
        Recording:
          InactiveToActive = TRUE
          UnacknowledgedToAcknowledged = TRUE
          AcknowledgedToUnacknowledged = FALSE
          UnconfirmedToConfirmed = TRUE
          ConfirmedToUnconfirmed = FALSE
          Update = FALSE
        Monitoring:
          MonitoredPV = ::AlarmX:Loc.Status.Alerts.Single.Stop[9]
          TriggerValues:
            [0] = 1
          Settings = 0
            Delay = 0.0
      Disable = FALSE
      InhibitPV
      AdditionalInformation1
      AdditionalInformation2
    [10]:
      Name = Alert.10
      Message = {$AlarmX/Alerts/Alert.10}
      Code = 10
      Severity = 2
      Behavior = DiscreteValueMonitoring
        Confirm = 0
        ReactionWhilePending = TRUE
        Recording:
          InactiveToActive = TRUE
          UnacknowledgedToAcknowledged = TRUE
          AcknowledgedToUnacknowledged = FALSE
          UnconfirmedToConfirmed = TRUE
          ConfirmedToUnconfirmed = FALSE
          Update = FALSE
        Monitoring:
          MonitoredPV = ::AlarmX:Loc.Status.Alerts.Single.Stop[10]
          TriggerValues:
            [0] = 1
          Settings = 0
            Delay = 0.0
      Disable = FALSE
      InhibitPV
      AdditionalInformation1
      AdditionalInformation2
    [11]:
      Name = Alert.11
      Message = {$AlarmX/Alerts/Alert.11}
      Code = 11
      Severity = 2
      Behavior = DiscreteValueMonitoring
        Confirm = 0
        ReactionWhilePending = TRUE
        Recording:
          InactiveToActive = TRUE
          UnacknowledgedToAcknowledged = TRUE
          AcknowledgedToUnacknowledged = FALSE
          UnconfirmedToConfirmed = TRUE
          ConfirmedToUnconfirmed = FALSE
          Update = FALSE
        Monitoring:
          MonitoredPV = ::AlarmX:Loc.Status.Alerts.Single.Stop[11]
          TriggerValues:
            [0] = 1
          Settings = 0
            Delay = 0.0
      Disable = FALSE
      InhibitPV
      AdditionalInformation1
      AdditionalInformation2
    [12]:
      Name = Alert.950
      Message = {$AlarmX/Alerts/Alert.950}
      Code = 1000
      Severity = 3
      Behavior = DiscreteValueMonitoring
        Confirm = 0
        ReactionWhilePending = TRUE
        Recording:
          InactiveToActive = TRUE
          UnacknowledgedToAcknowledged = TRUE
          AcknowledgedToUnacknowledged = FALSE
          UnconfirmedToConfirmed = TRUE
          ConfirmedToUnconfirmed = FALSE
          Update = FALSE
        Monitoring:
          MonitoredPV = ::AlarmX:Loc.Status.Alerts.Single.Info[950]
          TriggerValues:
            [0] = 1
          Settings = 0
            Delay = 0.0
      Disable = FALSE
      InhibitPV
      AdditionalInformation1
      AdditionalInformation2
    [13]:
      Name = Alert.1000
      Message = {$AlarmX/Alerts/Alert.1000}
      Code = 1000
      Severity = 3
      Behavior = DiscreteValueMonitoring
        Confirm = 0
        ReactionWhilePending = TRUE
        Recording:
          InactiveToActive = TRUE
          UnacknowledgedToAcknowledged = TRUE
          AcknowledgedToUnacknowledged = FALSE
          UnconfirmedToConfirmed = TRUE
          ConfirmedToUnconfirmed = FALSE
          Update = FALSE
        Monitoring:
          MonitoredPV = ::AlarmX:Loc.Status.Alerts.Single.Info[1000]
          TriggerValues:
            [0] = 1
          Settings = 0
            Delay = 0.0
      Disable = FALSE
      InhibitPV
      AdditionalInformation1
      AdditionalInformation2
    [14]:
      Name = Alert.1001
      Message = {$AlarmX/Alerts/Alert.1001}
      Code = 1001
      Severity = 3
      Behavior = DiscreteValueMonitoring
        Confirm = 0
        ReactionWhilePending = TRUE
        Recording:
          InactiveToActive = TRUE
          UnacknowledgedToAcknowledged = TRUE
          AcknowledgedToUnacknowledged = FALSE
          UnconfirmedToConfirmed = TRUE
          ConfirmedToUnconfirmed = FALSE
          Update = FALSE
        Monitoring:
          MonitoredPV = ::AlarmX:Loc.Status.Alerts.Single.Info[1001]
          TriggerValues:
            [0] = 1
          Settings = 0
            Delay = 0.0
      Disable = FALSE
      InhibitPV
      AdditionalInformation1
      AdditionalInformation2
    [15]:
      Name = Alert.1002
      Message = {$AlarmX/Alerts/Alert.1002}
      Code = 1002
      Severity = 3
      Behavior = DiscreteValueMonitoring
        Confirm = 0
        ReactionWhilePending = TRUE
        Recording:
          InactiveToActive = TRUE
          UnacknowledgedToAcknowledged = TRUE
          AcknowledgedToUnacknowledged = FALSE
          UnconfirmedToConfirmed = TRUE
          ConfirmedToUnconfirmed = FALSE
          Update = FALSE
        Monitoring:
          MonitoredPV = ::AlarmX:Loc.Status.Alerts.Single.Info[1002]
          TriggerValues:
            [0] = 1
          Settings = 0
            Delay = 0.0
      Disable = FALSE
      InhibitPV
      AdditionalInformation1
      AdditionalInformation2
    [16]:
      Name = Alert.1003
      Message = {$AlarmX/Alerts/Alert.1003}
      Code = 1003
      Severity = 3
      Behavior = DiscreteValueMonitoring
        Confirm = 0
        ReactionWhilePending = TRUE
        Recording:
          InactiveToActive = TRUE
          UnacknowledgedToAcknowledged = TRUE
          AcknowledgedToUnacknowledged = FALSE
          UnconfirmedToConfirmed = TRUE
          ConfirmedToUnconfirmed = FALSE
          Update = FALSE
        Monitoring:
          MonitoredPV = ::AlarmX:Loc.Status.Alerts.Single.Info[1003]
          TriggerValues:
            [0] = 1
          Settings = 0
            Delay = 0.0
      Disable = FALSE
      InhibitPV
      AdditionalInformation1
      AdditionalInformation2
    [17]:
      Name = Alert.1004
      Message = {$AlarmX/Alerts/Alert.1003}
      Code = 1004
      Severity = 3
      Behavior = DiscreteValueMonitoring
        Confirm = 0
        ReactionWhilePending = TRUE
        Recording:
          InactiveToActive = TRUE
          UnacknowledgedToAcknowledged = TRUE
          AcknowledgedToUnacknowledged = FALSE
          UnconfirmedToConfirmed = TRUE
          ConfirmedToUnconfirmed = FALSE
          Update = FALSE
        Monitoring:
          MonitoredPV = ::AlarmX:Loc.Status.Alerts.Single.Info[1003]
          TriggerValues:
            [0] = 1
          Settings = 0
            Delay = 0.0
      Disable = FALSE
      InhibitPV
      AdditionalInformation1
      AdditionalInformation2
    [18]:
      Name = Alert.1005
      Message = {$AlarmX/Alerts/Alert.1005}
      Code = 1005
      Severity = 3
      Behavior = DiscreteValueMonitoring
        Confirm = 0
        ReactionWhilePending = TRUE
        Recording:
          InactiveToActive = TRUE
          UnacknowledgedToAcknowledged = TRUE
          AcknowledgedToUnacknowledged = FALSE
          UnconfirmedToConfirmed = TRUE
          ConfirmedToUnconfirmed = FALSE
          Update = FALSE
        Monitoring:
          MonitoredPV = ::AlarmX:Loc.Status.Alerts.Single.Info[1005]
          TriggerValues:
            [0] = 1
          Settings = 0
            Delay = 0.0
      Disable = FALSE
      InhibitPV
      AdditionalInformation1
      AdditionalInformation2
    [19]:
      Name = Alert.1006
      Message = {$AlarmX/Alerts/Alert.1006}
      Code = 1006
      Severity = 3
      Behavior = DiscreteValueMonitoring
        Confirm = 0
        ReactionWhilePending = TRUE
        Recording:
          InactiveToActive = TRUE
          UnacknowledgedToAcknowledged = TRUE
          AcknowledgedToUnacknowledged = FALSE
          UnconfirmedToConfirmed = TRUE
          ConfirmedToUnconfirmed = FALSE
          Update = FALSE
        Monitoring:
          MonitoredPV = ::AlarmX:Loc.Status.Alerts.Single.Info[1006]
          TriggerValues:
            [0] = 1
          Settings = 0
            Delay = 0.0
      Disable = FALSE
      InhibitPV
      AdditionalInformation1
      AdditionalInformation2
    [20]:
      Name = Alert.1007
      Message = {$AlarmX/Alerts/Alert.1007}
      Code = 1007
      Severity = 3
      Behavior = DiscreteValueMonitoring
        Confirm = 0
        ReactionWhilePending = TRUE
        Recording:
          InactiveToActive = TRUE
          UnacknowledgedToAcknowledged = TRUE
          AcknowledgedToUnacknowledged = FALSE
          UnconfirmedToConfirmed = TRUE
          ConfirmedToUnconfirmed = FALSE
          Update = FALSE
        Monitoring:
          MonitoredPV = ::AlarmX:Loc.Status.Alerts.Single.Info[1007]
          TriggerValues:
            [0] = 1
          Settings = 0
            Delay = 0.0
      Disable = FALSE
      InhibitPV
      AdditionalInformation1
      AdditionalInformation2
    [21]:
      Name = Alert.1008
      Message = {$AlarmX/Alerts/Alert.1008}
      Code = 1008
      Severity = 3
      Behavior = DiscreteValueMonitoring
        Confirm = 0
        ReactionWhilePending = TRUE
        Recording:
          InactiveToActive = TRUE
          UnacknowledgedToAcknowledged = TRUE
          AcknowledgedToUnacknowledged = FALSE
          UnconfirmedToConfirmed = TRUE
          ConfirmedToUnconfirmed = FALSE
          Update = FALSE
        Monitoring:
          MonitoredPV = ::AlarmX:Loc.Status.Alerts.Single.Info[1008]
          TriggerValues:
            [0] = 1
          Settings = 0
            Delay = 0.0
      Disable = FALSE
      InhibitPV
      AdditionalInformation1
      AdditionalInformation2
    [22]:
      Name = Alert.1020
      Message = {$AlarmX/Alerts/Alert.1020}
      Code = 1002
      Severity = 3
      Behavior = DiscreteValueMonitoring
        Confirm = 0
        ReactionWhilePending = TRUE
        Recording:
          InactiveToActive = TRUE
          UnacknowledgedToAcknowledged = TRUE
          AcknowledgedToUnacknowledged = FALSE
          UnconfirmedToConfirmed = TRUE
          ConfirmedToUnconfirmed = FALSE
          Update = FALSE
        Monitoring:
          MonitoredPV = ::AlarmX:Loc.Status.Alerts.Single.Info[1020]
          TriggerValues:
            [0] = 1
          Settings = 0
            Delay = 0.0
      Disable = FALSE
      InhibitPV
      AdditionalInformation1
      AdditionalInformation2
    [23]:
      Name = Alert.1021
      Message = {$AlarmX/Alerts/Alert.1021}
      Code = 1002
      Severity = 3
      Behavior = DiscreteValueMonitoring
        Confirm = 0
        ReactionWhilePending = TRUE
        Recording:
          InactiveToActive = TRUE
          UnacknowledgedToAcknowledged = TRUE
          AcknowledgedToUnacknowledged = FALSE
          UnconfirmedToConfirmed = TRUE
          ConfirmedToUnconfirmed = FALSE
          Update = FALSE
        Monitoring:
          MonitoredPV = ::AlarmX:Loc.Status.Alerts.Single.Info[1021]
          TriggerValues:
            [0] = 1
          Settings = 0
            Delay = 0.0
      Disable = FALSE
      InhibitPV
      AdditionalInformation1
      AdditionalInformation2
    [24]:
      Name = Alert.1022
      Message = {$AlarmX/Alerts/Alert.1022}
      Code = 1022
      Severity = 3
      Behavior = DiscreteValueMonitoring
        Confirm = 0
        ReactionWhilePending = TRUE
        Recording:
          InactiveToActive = TRUE
          UnacknowledgedToAcknowledged = TRUE
          AcknowledgedToUnacknowledged = FALSE
          UnconfirmedToConfirmed = TRUE
          ConfirmedToUnconfirmed = FALSE
          Update = FALSE
        Monitoring:
          MonitoredPV = ::AlarmX:Loc.Status.Alerts.Single.Info[1022]
          TriggerValues:
            [0] = 1
          Settings = 0
            Delay = 0.0
      Disable = FALSE
      InhibitPV
      AdditionalInformation1
      AdditionalInformation2
    [25]:
      Name = Alert.1023
      Message = {$AlarmX/Alerts/Alert.1023}
      Code = 1002
      Severity = 3
      Behavior = DiscreteValueMonitoring
        Confirm = 0
        ReactionWhilePending = TRUE
        Recording:
          InactiveToActive = TRUE
          UnacknowledgedToAcknowledged = TRUE
          AcknowledgedToUnacknowledged = FALSE
          UnconfirmedToConfirmed = TRUE
          ConfirmedToUnconfirmed = FALSE
          Update = FALSE
        Monitoring:
          MonitoredPV = ::AlarmX:Loc.Status.Alerts.Single.Info[1023]
          TriggerValues:
            [0] = 1
          Settings = 0
            Delay = 0.0
      Disable = FALSE
      InhibitPV
      AdditionalInformation1
      AdditionalInformation2
    [26]:
      Name = Alert.1024
      Message = {$AlarmX/Alerts/Alert.1024}
      Code = 1024
      Severity = 3
      Behavior = DiscreteValueMonitoring
        Confirm = 0
        ReactionWhilePending = TRUE
        Recording:
          InactiveToActive = TRUE
          UnacknowledgedToAcknowledged = TRUE
          AcknowledgedToUnacknowledged = FALSE
          UnconfirmedToConfirmed = TRUE
          ConfirmedToUnconfirmed = FALSE
          Update = FALSE
        Monitoring:
          MonitoredPV = ::AlarmX:Loc.Status.Alerts.Single.Info[1024]
          TriggerValues:
            [0] = 1
          Settings = 0
            Delay = 0.0
      Disable = FALSE
      InhibitPV
      AdditionalInformation1
      AdditionalInformation2
    [27]:
      Name = Alert.1025
      Message = {$AlarmX/Alerts/Alert.1025}
      Code = 1025
      Severity = 3
      Behavior = DiscreteValueMonitoring
        Confirm = 0
        ReactionWhilePending = TRUE
        Recording:
          InactiveToActive = TRUE
          UnacknowledgedToAcknowledged = TRUE
          AcknowledgedToUnacknowledged = FALSE
          UnconfirmedToConfirmed = TRUE
          ConfirmedToUnconfirmed = FALSE
          Update = FALSE
        Monitoring:
          MonitoredPV = ::AlarmX:Loc.Status.Alerts.Single.Info[1025]
          TriggerValues:
            [0] = 1
          Settings = 0
            Delay = 0.0
      Disable = FALSE
      InhibitPV
      AdditionalInformation1
      AdditionalInformation2
  mapp.AlarmX.Snippets:
    AutoDetect = 1
      Language
    [0]:
      Key = TextSnippet.0
      Value = PV
        PV = ::gTextSnippet[0]
      Alarm
    [1]:
      Key = TextSnippet.1
      Value = PV
        PV = ::gTextSnippet[1]
      Alarm
    [2]:
      Key = TextSnippet.2
      Value = PV
        PV = ::gTextSnippet[2]
      Alarm
    [3]:
      Key = TextSnippet.3
      Value = PV
        PV = ::gTextSnippet[3]
      Alarm
    [4]:
      Key = TextSnippet.4
      Value = PV
        PV = ::gTextSnippet[4]
      Alarm
    [5]:
      Key = TextSnippet.5
      Value = PV
        PV = ::gTextSnippet[5]
      Alarm
```

- AlmXLStop.mpalarmxlist (1705107 bytes, not shown)

### Config_1.mpfilemanager - X20CP1685/mappServices/Config_1.mpfilemanager
```
Element FileManagement (Type=mpfilemanager)
  mapp.Gen:
    Enable = TRUE
    EnableCockpit = TRUE
    Audit = TRUE
    Parent
  FileManager:
    USB = 0
    Devices:
      0:
        DeviceName = DEV_CNC
        Text = DEVICE_CNC
    Access:
      0:
        Folder = *
```

### SyncModule.mppackmlsynchronizedmodule - X20CP1685/mappServices/PML/SyncModule.mppackmlsynchronizedmodule
```
Element gMpLink_PackMLSyncModule_CncCtrl (Type=mppackmlsynchronizedmodule)
  mapp.Gen:
    Enable = TRUE
    EnableCockpit = TRUE
    TaskClass = 1
    Auditing = MpAudit
      AuditStateDescription = 0
  Module:
    Name = CncCtrl
    Parent = 1
      Unit = gMpLink_PackMLSyncUnit_CORE
      Activation = 0
```

### SyncUnit.mppackmlsynchronizedunit - X20CP1685/mappServices/PML/SyncUnit.mppackmlsynchronizedunit
```
Element gMpLink_PackMLSyncUnit_CORE (Type=mppackmlsynchronizedunit)
  Settings:
    StartupActiveMode = 1
    BlockingModule
    StarvingModule
    AbortedByModule
    WaitingForModule
    ResetCommands = 1
  Modes:
    Mode[1]:
      ModeID = 1
      Name = Mode[3]
      State[2]:
        ChangeModeAllowed = TRUE
        StateCompleteRequired = FALSE
      State[3]:
        StateCompleteRequiredForStop = TRUE
      State[4]:
        ChangeModeAllowed = FALSE
        StateCompleteRequired = FALSE
      State[5]:
        ChangeModeAllowed = FALSE
        StateCompleteRequired = FALSE
        State[13]:
          StateCompleteRequiredForStop = TRUE
        State[14]:
          StateCompleteRequiredForStop = TRUE
      State[6]:
        ChangeModeAllowed = FALSE
        StateCompleteRequired = FALSE
      State[9]:
        ChangeModeAllowed = FALSE
        StateCompleteRequired = FALSE
      State[11]:
        ChangeModeAllowed = FALSE
        StateCompleteRequired = FALSE
        State[10]:
          StateCompleteRequiredForStop = TRUE
        State[12]:
          StateCompleteRequiredForStop = TRUE
      State[15]:
        StateCompleteRequiredForStop = TRUE
      State[17]:
        ChangeModeAllowed = FALSE
        StateCompleteRequired = FALSE
        State[16]:
          StateCompleteRequiredForStop = TRUE
      State[31]:
        ChangeModeAllowed = FALSE
        StateCompleteRequired = FALSE
    Mode[2]:
      ModeID = 2
      Name = Production
      State[2]:
        ChangeModeAllowed = TRUE
        StateCompleteRequired = FALSE
      State[3]:
        StateCompleteRequiredForStop = TRUE
      State[4]:
        ChangeModeAllowed = FALSE
        StateCompleteRequired = FALSE
      State[5]:
        ChangeModeAllowed = FALSE
        StateCompleteRequired = FALSE
        State[13]:
          StateCompleteRequiredForStop = TRUE
        State[14]:
          StateCompleteRequiredForStop = TRUE
      State[6]:
        ChangeModeAllowed = FALSE
        StateCompleteRequired = FALSE
      State[9]:
        ChangeModeAllowed = FALSE
        StateCompleteRequired = FALSE
      State[11]:
        ChangeModeAllowed = FALSE
        StateCompleteRequired = FALSE
        State[10]:
          StateCompleteRequiredForStop = TRUE
        State[12]:
          StateCompleteRequiredForStop = TRUE
      State[15]:
        StateCompleteRequiredForStop = TRUE
      State[17]:
        ChangeModeAllowed = FALSE
        StateCompleteRequired = FALSE
        State[16]:
          StateCompleteRequiredForStop = TRUE
      State[31]:
        ChangeModeAllowed = FALSE
        StateCompleteRequired = FALSE
    Mode[3]:
      ModeID = 3
      Name = Mode[2]
      State[2]:
        ChangeModeAllowed = TRUE
        StateCompleteRequired = FALSE
      State[3]:
        StateCompleteRequiredForStop = TRUE
      State[4]:
        ChangeModeAllowed = FALSE
        StateCompleteRequired = FALSE
      State[5]:
        ChangeModeAllowed = FALSE
        StateCompleteRequired = FALSE
        State[13]:
          StateCompleteRequiredForStop = TRUE
        State[14]:
          StateCompleteRequiredForStop = TRUE
      State[6]:
        ChangeModeAllowed = FALSE
        StateCompleteRequired = FALSE
      State[9]:
        ChangeModeAllowed = FALSE
        StateCompleteRequired = FALSE
      State[11]:
        ChangeModeAllowed = FALSE
        StateCompleteRequired = FALSE
        State[10]:
          StateCompleteRequiredForStop = TRUE
        State[12]:
          StateCompleteRequiredForStop = TRUE
      State[15]:
        StateCompleteRequiredForStop = TRUE
      State[17]:
        ChangeModeAllowed = FALSE
        StateCompleteRequired = FALSE
        State[16]:
          StateCompleteRequiredForStop = TRUE
      State[31]:
        ChangeModeAllowed = FALSE
        StateCompleteRequired = FALSE
```

### UsrXLogin.mpuserxlogin - X20CP1685/mappServices/UserX/UsrXLogin.mpuserxlogin
```
Element gMpLink_UserXLogin (Type=mpuserxlogin)
  mapp.Gen:
    Enable = TRUE
    EnableCockpit = TRUE
    Audit = TRUE
    Parent
```

## Logical view

Binary libraries used (declarations not repeated): operator, runtime, AsIecCon, astime, FileIO, AsBrStr, standard, sys_lib, AsZip, MpBase, McBase 6.7.2, MpAxis 6.7.2, McAcpAx 6.7.2, McPathGen 6.7.2, McAcpTrak 6.7.2, McAxGroup 6.7.2, McAxis 6.7.2, McProgInt 6.7.2, MpRecipe 6.7.1, MpUserX 6.7.1, MpCnc 6.7.2, MpFile 6.7.1, MpPackML 6.7.1, MpAlarmX 6.7.1, CoTrace 6.7.0, MpServer 6.5.0, McPureVAx 6.7.2

### Package Logical/Libraries - Global libraries

### Library Logical/Libraries/aLibFile (IEC, version 1.0.0) - Bu yapı içerisinde file/folder oluşturma, bunlara yazma, silme gibi fb ler mevcut.
Depends on: FileIO, AsBrStr, standard

#### Notes.txt
```
(* PC de veya CPU da 'C' ye oluşturur *)
FB_DirCreate.Parameters.DeviceName := 'Device_CNCprg';
FB_DirCreate.Parameters.DirPath := '/DEVICE=X:\\CNCPrg\';

(* PLC altındaki F ye oluşturur - windows suzlarda *)
FB_DirCreate.Parameters.DeviceName := 'Device_RECIPE';
FB_DirCreate.Parameters.DirPath := '/DEVICE=USER_PATH/Recipe';
```

#### FbDirCreate.typ - Exported data types
```iecst
(********************************************************************
 * COPYRIGHT --  B&R Industrial Automation GmbH
 *******************************************************************
 * Library: aLibFile
 * Function Block: FbDirCreate
 * Author: kay3a
 * Created: August 27, 2024/4:57 PM
 ********************************************************************)
(**)
(**** FB Parameters Type*)

TYPE
	Par_DirCreate_typ : 	STRUCT  (**** FB Parameters Type*)
		DeviceName : STRING[80]; (*- Istenilen essiz device name parametresi. ex: "Device_deneme"*)
		DirPath : STRING[80]; (*- Folder olmasi istenilen direction. ex: "/DEVICE=USER_PATH/deneme/" yada "/DEVICE=C:\\deneme/"  gibi.*)
	END_STRUCT;
END_TYPE

(**)
(**)
(**)
(**)
(**** Internal Type*)

TYPE
	Int_DirCreate_typ : 	STRUCT  (**** Internal Type*)
		Step : Int_DirCreate_Step_enum; (*- Proses case steps.*)
		FB : Int_DirCreate_FB_typ; (*- Internal usage FBs.*)
		CapturedExecute : BOOL; (*- Execute istegi yakalandi flagi.*)
	END_STRUCT;
END_TYPE

(**)
(**** Internal FB Type*)

TYPE
	Int_DirCreate_FB_typ : 	STRUCT  (**** Internal FB Type*)
		_DirCreate : DirCreate; (*- Folder olusturmak için B&R fb.*)
		_DevLink : DevLink; (*- Device olusturmak için B&R fb.*)
	END_STRUCT;
END_TYPE

(**)
(**** Internal Step Enum Type*)

TYPE
	Int_DirCreate_Step_enum :
		( (**** Internal Step Enum Type*)
		stepDirCreate_0_Idle := 0, (*- FB idle.*)
		stepDirCreate_1_WaitCmd := 1, (*- Yeni komut için hazir step.*)
		stepDirCreate_2_CrateDevLink := 2, (*- Device olusturma step.*)
		stepDirCreate_3_CreateDir := 3, (*- Folder olusturma step.*)
		stepDirCreate_10_Done := 10, (*- Islem basariyla tamamlandi step.*)
		stepDirCreate_11_Error := 11 (*- Error step.*)
		);
END_TYPE
```

#### FbDirDelete.typ - Exported data types
```iecst
(********************************************************************
 * COPYRIGHT --  B&R Industrial Automation GmbH
 *******************************************************************
 * Library: aLibFile
 * Function Block: FbDirDelete
 * Author: kay3a
 * Created: August 27, 2024/4:57 PM
 ********************************************************************)
(**)
(**** FB Parameters Type*)

TYPE
	Par_DirDelete_typ : 	STRUCT  (**** FB Parameters Type*)
		DeviceName : STRING[80]; (*- Istenilen essiz device name parametresi. ex: "Device_deneme"*)
	END_STRUCT;
END_TYPE

(**)
(**)
(**)
(**)
(**** Internal Type*)

TYPE
	Int_DirDelete_typ : 	STRUCT  (**** Internal Type*)
		Step : Int_DirDelete_Step_enum; (*- Proses case steps.*)
		FB : Int_DirDelete_FB_typ; (*- Internal usage FBs.*)
		CapturedExecute : BOOL; (*- Execute istegi yakalandi flagi.*)
	END_STRUCT;
END_TYPE

(**)
(**** Internal FB Type*)

TYPE
	Int_DirDelete_FB_typ : 	STRUCT  (**** Internal FB Type*)
		_DirDelete : DirDeleteEx; (*- Folder silmek için B&R fb.*)
	END_STRUCT;
END_TYPE

(**)
(**** Internal Step Enum Type*)

TYPE
	Int_DirDelete_Step_enum :
		( (**** Internal Step Enum Type*)
		stepDirDelete_0_Idle := 0, (*- FB idle.*)
		stepDirDelete_1_WaitCmd := 1, (*- Yeni komut için hazir step.*)
		stepDirDelete_2_Delete := 2, (*- Folder silme step.*)
		stepDirDelete_10_Done := 10, (*- Islem basariyla tamamlandi step.*)
		stepDirDelete_11_Error := 11 (*- Error step.*)
		);
END_TYPE
```

#### FbDirRead.typ - Exported data types
```iecst
(********************************************************************
 * COPYRIGHT --  B&R Industrial Automation GmbH
 *******************************************************************
 * Library: aLibFile
 * Function Block: FbDirRead
 * Author: kay3a
 * Created: August 27, 2024/4:57 PM
 ********************************************************************)
(**)
(**** FB Parameters Type*)

TYPE
	Par_DirRead_typ : 	STRUCT  (**** FB Parameters Type*)
		DeviceName : STRING[80]; (*- Istenilen essiz device name parametresi. ex: "Device_deneme"*)
	END_STRUCT;
END_TYPE

(**)
(**)
(**)
(**)
(**** Internal Type*)

TYPE
	Int_DirRead_typ : 	STRUCT  (**** Internal Type*)
		Step : Int_DirRead_Step_enum; (*- Proses case steps.*)
		CountFile : UDINT; (*- Okuma esnasinda sayma degiskeni.*)
		ReadFile : fiDIR_READ_EX_DATA; (*- Okuma tipi.*)
		FB : Int_DirRead_FB_typ; (*- Internal usage FBs.*)
		CapturedExecute : BOOL; (*- Execute istegi yakalandi flagi.*)
	END_STRUCT;
END_TYPE

(**)
(**** Internal FB Type*)

TYPE
	Int_DirRead_FB_typ : 	STRUCT  (**** Internal FB Type*)
		_DirInfo : DirInfo; (*- Folder bilgisi almak için B&R fb.*)
		_DirRead : DirRead; (*- Folder içindekileri okuyup siralamak için B&R fb.*)
	END_STRUCT;
END_TYPE

(**)
(**** Internal Step Enum Type*)

TYPE
	Int_DirRead_Step_enum :
		( (**** Internal Step Enum Type*)
		stepDirRead_0_Idle := 0, (*- FB idle.*)
		stepDirRead_1_WaitCmd := 1, (*- Yeni komut için hazir step.*)
		stepDirRead_2_GetInfo := 2, (*- Folder info alma step.*)
		stepDirRead_3_Read := 3, (*- Folder içini okuma step.*)
		stepDirRead_10_Done := 10, (*- Islem basariyla tamamlandi step.*)
		stepDirRead_11_Error := 11 (*- Error step.*)
		);
END_TYPE
```

#### FbFileCreate.typ - Exported data types
```iecst
(********************************************************************
 * COPYRIGHT --  B&R Industrial Automation GmbH
 *******************************************************************
 * Library: aLibFile
 * Function Block: FbFileCreate
 * Author: kay3a
 * Created: August 27, 2024/4:57 PM
 ********************************************************************)
(**)
(**** FB Parameters Type*)

TYPE
	Par_FileCreate_typ : 	STRUCT  (**** FB Parameters Type*)
		DeviceName : STRING[80]; (*- Istenilen essiz device name parametresi. ex: "Device_deneme"*)
		FileName : STRING[80]; (*- Istenilen folder içerisinde olusturulacak File ismi.*)
	END_STRUCT;
END_TYPE

(**)
(**)
(**)
(**)
(**** Internal Type*)

TYPE
	Int_FileCreate_typ : 	STRUCT  (**** Internal Type*)
		Step : Int_FileCreate_Step_enum; (*- Proses case steps.*)
		FB : Int_FileCreate_FB_typ; (*- Internal usage FBs.*)
		CapturedExecute : BOOL; (*- Execute istegi yakalandi flagi.*)
	END_STRUCT;
END_TYPE

(**)
(**** Internal FB Type*)

TYPE
	Int_FileCreate_FB_typ : 	STRUCT  (**** Internal FB Type*)
		_FileCreate : FileCreate; (*- File olusturmak için B&R fb.*)
		_FileClose : FileClose; (*- File kapatmak için B&R fb.*)
	END_STRUCT;
END_TYPE

(**)
(**** Internal Step Enum Type*)

TYPE
	Int_FileCreate_Step_enum :
		( (**** Internal Step Enum Type*)
		stepFileCreate_0_Idle := 0, (*- FB idle.*)
		stepFileCreate_1_WaitCmd := 1, (*- Yeni komut için hazir step.*)
		stepFileCreate_2_Create := 2, (*- File olusturma step.*)
		stepFileCreate_3_Close := 3, (*- File kapatma step.*)
		stepFileCreate_10_Done := 10, (*- Islem basariyla tamamlandi step.*)
		stepFileCreate_11_Error := 11 (*- Error step.*)
		);
END_TYPE
```

#### FbFileWrite.typ - Exported data types
```iecst
(********************************************************************
 * COPYRIGHT --  B&R Industrial Automation GmbH
 *******************************************************************
 * Library: aLibFile
 * Function Block: FbFileWrite
 * Author: kay3a
 * Created: August 27, 2024/4:57 PM
 ********************************************************************)
(**)
(**** FB Parameters Type*)

TYPE
	Par_FileWrite_typ : 	STRUCT  (**** FB Parameters Type*)
		DeviceName : STRING[80]; (*- Istenilen essiz device name parametresi. ex: "Device_deneme"*)
		FileName : STRING[80]; (*- Folder içerisinde içerisine yazilmak istenilen file ismi.*)
	END_STRUCT;
END_TYPE

(**)
(**)
(**)
(**)
(**** Internal Type*)

TYPE
	Int_FileWrite_typ : 	STRUCT  (**** Internal Type*)
		Step : Int_FileWrite_Step_enum; (*- Proses case steps.*)
		FB : Int_FileWrite_FB_typ; (*- Internal usage FBs.*)
		CapturedExecute : BOOL; (*- Execute istegi yakalandi flagi.*)
	END_STRUCT;
END_TYPE

(**)
(**** Internal FB Type*)

TYPE
	Int_FileWrite_FB_typ : 	STRUCT  (**** Internal FB Type*)
		_FileOpen : FileOpen; (*- File açmak için B&R fb.*)
		_FileWriteEx : FileWriteEx; (*- File yazmak için B&R fb.*)
		_FileClose : FileClose; (*- File kapatmak için B&R fb.*)
	END_STRUCT;
END_TYPE

(**)
(**** Internal Step Enum Type*)

TYPE
	Int_FileWrite_Step_enum :
		( (**** Internal Step Enum Type*)
		stepFileWrite_0_Idle := 0, (*- FB idle.*)
		stepFileWrite_1_WaitCmd := 1, (*- Yeni komut için hazir step.*)
		stepFileWrite_2_FileOpen := 2, (*- File açma step.*)
		stepFileWrite_3_Write := 3, (*- File yazma step.*)
		stepFileWrite_4_FileClose := 4, (*- File kapatma step.*)
		stepFileWrite_10_Done := 10, (*- Islem basariyla tamamlandi step.*)
		stepFileWrite_11_Error := 11 (*- Error step.*)
		);
END_TYPE
```

#### FbFileRead.typ - Exported data types
```iecst
(********************************************************************
 * COPYRIGHT --  B&R Industrial Automation GmbH
 *******************************************************************
 * Library: aLibFile
 * Function Block: FbFileRead
 * Author: kay3a
 * Created: August 27, 2024/4:57 PM
 ********************************************************************)
(**)
(**** FB Parameters Type*)

TYPE
	Par_FileRead_typ : 	STRUCT  (**** FB Parameters Type*)
		DeviceName : STRING[80]; (*- Istenilen essiz device name parametresi. ex: "Device_deneme"*)
		FileName : STRING[80]; (*- Folder içerisinde içerisine okunmak istenilen file ismi.*)
	END_STRUCT;
END_TYPE

(**)
(**)
(**)
(**)
(**** Internal Type*)

TYPE
	Int_FileRead_typ : 	STRUCT  (**** Internal Type*)
		Step : Int_FileRead_Step_enum; (*- Proses case steps.*)
		FB : Int_FileRead_FB_typ; (*- Internal usage FBs.*)
		CapturedExecute : BOOL; (*- Execute istegi yakalandi flagi.*)
	END_STRUCT;
END_TYPE

(**)
(**** Internal FB Type*)

TYPE
	Int_FileRead_FB_typ : 	STRUCT  (**** Internal FB Type*)
		_FileOpen : FileOpen; (*- File açmak için B&R fb.*)
		_FileReadEx : FileReadEx; (*- File okumak için B&R fb.*)
		_FileClose : FileClose; (*- File kapatmak için B&R fb.*)
	END_STRUCT;
END_TYPE

(**)
(**** Internal Step Enum Type*)

TYPE
	Int_FileRead_Step_enum :
		( (**** Internal Step Enum Type*)
		stepFileRead_0_Idle := 0, (*- FB idle.*)
		stepFileRead_1_WaitCmd := 1, (*- Yeni komut için hazir step.*)
		stepFileRead_2_FileOpen := 2, (*- File açma step.*)
		stepFileRead_3_Read := 3, (*- File okuma step.*)
		stepFileRead_4_FileClose := 4, (*- File kapatma step.*)
		stepFileRead_10_Done := 10, (*- Islem basariyla tamamlandi step.*)
		stepFileRead_11_Error := 11 (*- Error step.*)
		);
END_TYPE
```

#### FbFileDelete.typ - Exported data types
```iecst
(********************************************************************
 * COPYRIGHT --  B&R Industrial Automation GmbH
 *******************************************************************
 * Library: aLibFile
 * Function Block: FbFileDelete
 * Author: kay3a
 * Created: August 27, 2024/4:57 PM
 ********************************************************************)
(**)
(**** FB Parameters Type*)

TYPE
	Par_FileDelete_typ : 	STRUCT  (**** FB Parameters Type*)
		DeviceName : STRING[80]; (*- Istenilen essiz device name parametresi. ex: "Device_deneme"*)
		FileName : STRING[80]; (*- Seçili folder içerisinden silinmek istenilen file.*)
	END_STRUCT;
END_TYPE

(**)
(**)
(**)
(**)
(**** Internal Type*)

TYPE
	Int_FileDelete_typ : 	STRUCT  (**** Internal Type*)
		Step : Int_FileDelete_Step_enum; (*- Proses case steps.*)
		FB : Int_FileDelete_FB_typ; (*- Internal usage FBs.*)
		CapturedExecute : BOOL; (*- Execute istegi yakalandi flagi.*)
	END_STRUCT;
END_TYPE

(**)
(**** Internal FB Type*)

TYPE
	Int_FileDelete_FB_typ : 	STRUCT  (**** Internal FB Type*)
		_FileDelete : FileDelete; (*- File silmek için B&R fb.*)
	END_STRUCT;
END_TYPE

(**)
(**** Internal Step Enum Type*)

TYPE
	Int_FileDelete_Step_enum :
		( (**** Internal Step Enum Type*)
		stepFileDelete_0_Idle := 0, (*- FB idle.*)
		stepFileDelete_1_WaitCmd := 1, (*- Yeni komut için hazir step.*)
		stepFileDelete_2_Delete := 2, (*- File silme step.*)
		stepFileDelete_10_Done := 10, (*- Islem basariyla tamamlandi step.*)
		stepFileDelete_11_Error := 11 (*- Error step.*)
		);
END_TYPE
```

#### aLibFile.fun - Exported functions and function blocks
```iecst
(********************************************************************
 * COPYRIGHT --  B&R Industrial Automation GmbH
 *******************************************************************
 * Library: myLibFile
 * Author: kay3a
 * Created: August 27, 2024/4:53 PM
 *******************************************************************
 * Description: Bu Library içerisinde file/ folder ile ilgili
                       ihtiyaç duydugunuz birçok islemi yapabileceginiz
                       FB ler mevcut.
 ********************************************************************)

{REDUND_ERROR} FUNCTION_BLOCK FbDirDelete (*- Folder silme FB.*) (*$GROUP=User,$CAT=User,$GROUPICON=User.png,$CATICON=User.png*)
	VAR_INPUT
		Enable : BOOL; (*- FB Enable.*)
		Execute : BOOL; (*- FB Execute cmd.*)
		ErrorReset : BOOL; (*- FB ErrorReset cmd.*)
		Parameters : Par_DirDelete_typ; (*- FB Parameters.*)
	END_VAR
	VAR_OUTPUT
		Active : BOOL; (*- FB Activated.*)
		CommandBusy : BOOL; (*- FB CommandBusy flag.*)
		CommandDone : BOOL; (*- FB CommandDone flag.*)
		Error : BOOL; (*- FB Error flag.*)
		StatusID : DINT; (*- FB Error Status ID.*)
	END_VAR
	VAR
		Internal : Int_DirDelete_typ; (*- FB Internal variables.*)
		zzEdge00000 : BOOL;
	END_VAR
END_FUNCTION_BLOCK

{REDUND_ERROR} FUNCTION_BLOCK FbDirRead (*- Folder içindekileri okuma FB.*) (*$GROUP=User,$CAT=User,$GROUPICON=User.png,$CATICON=User.png*)
	VAR_INPUT
		Enable : BOOL; (*- Folder okuma FB.*)
		Execute : BOOL; (*- FB Execute cmd.*)
		ErrorReset : BOOL; (*- FB ErrorReset cmd.*)
		Parameters : Par_DirRead_typ; (*- FB Parameters.*)
	END_VAR
	VAR_OUTPUT
		Active : BOOL; (*- FB Activated.*)
		ListedFile : ARRAY[0..999] OF STRING[80]; (*- Listelenen file lar.*)
		CommandBusy : BOOL; (*- FB CommandBusy flag.*)
		CommandDone : BOOL; (*- FB CommandDone flag.*)
		Error : BOOL; (*- FB Error flag.*)
		StatusID : DINT; (*- FB Error Status ID.*)
	END_VAR
	VAR
		Internal : Int_DirRead_typ; (*- FB Internal variables.*)
		zzEdge00000 : BOOL;
	END_VAR
END_FUNCTION_BLOCK

{REDUND_ERROR} FUNCTION_BLOCK FbDirCreate (*- Folder olusturma FB.*) (*$GROUP=User,$CAT=User,$GROUPICON=User.png,$CATICON=User.png*)
	VAR_INPUT
		Enable : BOOL; (*- Folder olusturma FB.*)
		Execute : BOOL; (*- FB Execute cmd.*)
		ErrorReset : BOOL; (*- FB ErrorReset cmd.*)
		Parameters : Par_DirCreate_typ; (*- FB Parameters.*)
	END_VAR
	VAR_OUTPUT
		Active : BOOL; (*- FB Activated.*)
		CommandBusy : BOOL; (*- FB CommandBusy flag.*)
		CommandDone : BOOL; (*- FB CommandDone flag.*)
		Error : BOOL; (*- FB Error flag.*)
		StatusID : DINT; (*- FB Error Status ID.*)
	END_VAR
	VAR
		Internal : Int_DirCreate_typ; (*- FB Internal variables.*)
		zzEdge00000 : BOOL;
	END_VAR
END_FUNCTION_BLOCK

{REDUND_ERROR} FUNCTION_BLOCK FbFileCreate (*- Folder içerisine File olusturma FB.*) (*$GROUP=User,$CAT=User,$GROUPICON=User.png,$CATICON=User.png*)
	VAR_INPUT
		Enable : BOOL; (*- Folder olusturma FB.*)
		Execute : BOOL; (*- FB Execute cmd.*)
		ErrorReset : BOOL; (*- FB ErrorReset cmd.*)
		Parameters : Par_FileCreate_typ; (*- FB Parameters.*)
	END_VAR
	VAR_OUTPUT
		Active : BOOL; (*- FB Activated.*)
		CommandBusy : BOOL; (*- FB CommandBusy flag.*)
		CommandDone : BOOL; (*- FB CommandDone flag.*)
		Error : BOOL; (*- FB Error flag.*)
		StatusID : DINT; (*- FB Error Status ID.*)
	END_VAR
	VAR
		Internal : Int_FileCreate_typ; (*- FB Internal variables.*)
		zzEdge00000 : BOOL;
	END_VAR
END_FUNCTION_BLOCK

{REDUND_ERROR} FUNCTION_BLOCK FbFileWrite (*- File içine yazma FB.*) (*$GROUP=User,$CAT=User,$GROUPICON=User.png,$CATICON=User.png*)
	VAR_INPUT
		Enable : BOOL; (*- File içerisine yazma FB.*)
		Execute : BOOL; (*- FB Execute cmd.*)
		ErrorReset : BOOL; (*- FB ErrorReset cmd.*)
		Parameters : Par_FileWrite_typ; (*- FB Parameters.*)
		WriteData : STRING[99999]; (*- Okunan data.*)
	END_VAR
	VAR_OUTPUT
		Active : BOOL; (*- FB Activated.*)
		CommandBusy : BOOL; (*- FB CommandBusy flag.*)
		CommandDone : BOOL; (*- FB CommandDone flag.*)
		Error : BOOL; (*- FB Error flag.*)
		StatusID : DINT; (*- FB Error Status ID.*)
	END_VAR
	VAR
		Internal : Int_FileWrite_typ; (*- FB Internal variables.*)
		zzEdge00000 : BOOL;
	END_VAR
END_FUNCTION_BLOCK

{REDUND_ERROR} FUNCTION_BLOCK FbFileRead (*- File içerisini okuma FB.*) (*$GROUP=User,$CAT=User,$GROUPICON=User.png,$CATICON=User.png*)
	VAR_INPUT
		Enable : BOOL; (*- File içerisini okuma FB.*)
		Execute : BOOL; (*- FB Execute cmd.*)
		ErrorReset : BOOL; (*- FB ErrorReset cmd.*)
		Parameters : Par_FileRead_typ; (*- FB Parameters.*)
	END_VAR
	VAR_OUTPUT
		ReadData : STRING[99999]; (*- Okunan data.*)
		Active : BOOL; (*- FB Activated.*)
		CommandBusy : BOOL; (*- FB CommandBusy flag.*)
		CommandDone : BOOL; (*- FB CommandDone flag.*)
		Error : BOOL; (*- FB Error flag.*)
		StatusID : DINT; (*- FB Error Status ID.*)
	END_VAR
	VAR
		Internal : Int_FileRead_typ; (*- FB Internal variables.*)
		zzEdge00000 : BOOL;
	END_VAR
END_FUNCTION_BLOCK

{REDUND_ERROR} FUNCTION_BLOCK FbFileDelete (*- File silme FB.*) (*$GROUP=User,$CAT=User,$GROUPICON=User.png,$CATICON=User.png*)
	VAR_INPUT
		Enable : BOOL; (*- File silme FB.*)
		Execute : BOOL; (*- FB Execute cmd.*)
		ErrorReset : BOOL; (*- FB ErrorReset cmd.*)
		Parameters : Par_FileDelete_typ; (*- FB Parameters.*)
	END_VAR
	VAR_OUTPUT
		Active : BOOL; (*- FB Activated.*)
		CommandBusy : BOOL; (*- FB CommandBusy flag.*)
		CommandDone : BOOL; (*- FB CommandDone flag.*)
		Error : BOOL; (*- FB Error flag.*)
		StatusID : DINT; (*- FB Error Status ID.*)
	END_VAR
	VAR
		Internal : Int_FileDelete_typ; (*- FB Internal variables.*)
		zzEdge00000 : BOOL;
	END_VAR
END_FUNCTION_BLOCK
```

#### FbDirDelete.st - Folder siler.
```iecst
(********************************************************************
 * COPYRIGHT --  B&R Industrial Automation GmbH
 ********************************************************************
 * Library: aLibFile
 * Function Block: FbDirDelete
 * Author: kay3a
 * Created: August 27, 2024/4:58 PM
 ********************************************************************
 * Description: Bu FB parametreden girilen DeviceName deki folder silme islemini yapar.
********************************************************************)
FUNCTION_BLOCK FbDirDelete

	//|ŻŻŻŻŻŻŻŻŻŻŻŻŻŻŻŻŻŻŻŻŻŻŻŻŻŻŻŻŻŻŻŻŻŻŻŻŻŻŻŻŻŻŻŻŻŻŻŻŻŻŻŻŻŻŻŻŻŻŻŻŻŻŻŻŻŻŻŻŻŻŻŻŻ
	//|               FB ENABLE KONTROLU
	//|_________________________________________________________________________

	(* Enable gelirse FB aktiftir. Gelmiyorsa aktif degildir.  *)
	Active := Enable;

	(* Aktif degilse Step basa gelsin *)
	IF NOT Active THEN
		Internal.Step := stepDirDelete_0_Idle;
	END_IF;
	//|_________________________________________________________________________

	//|ŻŻŻŻŻŻŻŻŻŻŻŻŻŻŻŻŻŻŻŻŻŻŻŻŻŻŻŻŻŻŻŻŻŻŻŻŻŻŻŻŻŻŻŻŻŻŻŻŻŻŻŻŻŻŻŻŻŻŻŻŻŻŻŻŻŻŻŻŻŻŻŻŻ
	//|               CHECK FB ERROR
	//|_________________________________________________________________________

	(* Error check *)
	IF Internal.FB._DirDelete.enable AND (Internal.FB._DirDelete.status <> ERR_FUB_BUSY AND Internal.FB._DirDelete.status <> ERR_OK) THEN
		StatusID := Internal.FB._DirDelete.status;
		Internal.Step := stepDirDelete_11_Error;
	END_IF;
	//|_________________________________________________________________________

	//|ŻŻŻŻŻŻŻŻŻŻŻŻŻŻŻŻŻŻŻŻŻŻŻŻŻŻŻŻŻŻŻŻŻŻŻŻŻŻŻŻŻŻŻŻŻŻŻŻŻŻŻŻŻŻŻŻŻŻŻŻŻŻŻŻŻŻŻŻŻŻŻŻŻ
	//|               CHECK CMD FB EXECUTE
	//|_________________________________________________________________________

	(* Captured Execute *)
	IF EDGEPOS(Execute) THEN
		Internal.CapturedExecute := TRUE;
	ELSIF NOT Execute OR Error THEN
		Internal.CapturedExecute := FALSE;
	END_IF;
	//|_________________________________________________________________________

	//|=========================================================================
	//|					FILLING PROCESS STATE MACHINE
	//|
	//|
	//|=========================================================================
	CASE Internal.Step OF

		//=======================================================
		stepDirDelete_0_Idle: // Idle
			//=======================================================
			Error := FALSE;
			CommandDone := FALSE;
			CommandBusy := FALSE;
			IF Active THEN
				Internal.Step := stepDirDelete_1_WaitCmd;
			END_IF;
			//=======================================================

			//=======================================================
		stepDirDelete_1_WaitCmd: // Wait Cmd
			//=======================================================
			IF (Internal.CapturedExecute) THEN
				CommandBusy := TRUE;
				Internal.Step := stepDirDelete_2_Delete;
			END_IF;
			//=======================================================

			//=======================================================
		stepDirDelete_2_Delete: // Get Dir info
			//=======================================================
			(* Create folder for this component on the user file device *)
			Internal.FB._DirDelete.enable := TRUE;
			Internal.FB._DirDelete.pDevice := ADR(Parameters.DeviceName);
			Internal.FB._DirDelete.pName := ADR('\');
			Internal.FB._DirDelete();
			(* Check if folder already exist and if so disabled the function block call *)
			IF (Internal.FB._DirDelete.status = ERR_OK) THEN
				Internal.Step := stepDirDelete_10_Done;
			END_IF
			//=======================================================

			//=======================================================
		stepDirDelete_10_Done: // Done
			//=======================================================
			CommandDone := TRUE;
			IF NOT Execute THEN
				Internal.Step := stepDirDelete_0_Idle;
			END_IF;
			//=======================================================

			//=======================================================
		stepDirDelete_11_Error: // Error
			//=======================================================
			Error := TRUE;
			Internal.FB._DirDelete(enable := FALSE);
			IF ErrorReset THEN
				StatusID := ERR_OK;
				Internal.Step := stepDirDelete_0_Idle;
			END_IF;
		//=======================================================

	END_CASE;
	//|=========================================================================

END_FUNCTION_BLOCK
```

#### FbDirCreate.st - Folder oluşturur.
```iecst
(********************************************************************
 * COPYRIGHT --  B&R Industrial Automation GmbH
 ********************************************************************
 * Library: aLibFile
 * Function Block: FbDirCreate
 * Author: kay3a
 * Created: August 27, 2024/4:58 PM
 ********************************************************************
 * Description: Bu FB parametreden girilen DeviceName e folder olusturma islemini yapar.
 ********************************************************************)
FUNCTION_BLOCK FbDirCreate

	//|ŻŻŻŻŻŻŻŻŻŻŻŻŻŻŻŻŻŻŻŻŻŻŻŻŻŻŻŻŻŻŻŻŻŻŻŻŻŻŻŻŻŻŻŻŻŻŻŻŻŻŻŻŻŻŻŻŻŻŻŻŻŻŻŻŻŻŻŻŻŻŻŻŻ
	//|               FB ENABLE KONTROLU
	//|_________________________________________________________________________

	(* Enable gelirse FB aktiftir. Gelmiyorsa aktif degildir.  *)
	Active := Enable;

	(* Aktif degilse Step basa gelsin *)
	IF NOT Active THEN
		Internal.Step := stepDirCreate_0_Idle;
	END_IF;
	//|_________________________________________________________________________

	//|ŻŻŻŻŻŻŻŻŻŻŻŻŻŻŻŻŻŻŻŻŻŻŻŻŻŻŻŻŻŻŻŻŻŻŻŻŻŻŻŻŻŻŻŻŻŻŻŻŻŻŻŻŻŻŻŻŻŻŻŻŻŻŻŻŻŻŻŻŻŻŻŻŻ
	//|               CHECK FB ERROR
	//|_________________________________________________________________________

	(* Error check *)
	IF Internal.FB._DirCreate.enable AND (Internal.FB._DirCreate.status <> ERR_FUB_BUSY AND Internal.FB._DirCreate.status <> ERR_OK AND Internal.FB._DirCreate.status <> fiERR_DIR_ALREADY_EXIST) THEN
		StatusID := Internal.FB._DirCreate.status;
		Internal.Step := stepDirCreate_11_Error;
	END_IF;
	//|_________________________________________________________________________

	//|ŻŻŻŻŻŻŻŻŻŻŻŻŻŻŻŻŻŻŻŻŻŻŻŻŻŻŻŻŻŻŻŻŻŻŻŻŻŻŻŻŻŻŻŻŻŻŻŻŻŻŻŻŻŻŻŻŻŻŻŻŻŻŻŻŻŻŻŻŻŻŻŻŻ
	//|               CHECK CMD FB EXECUTE
	//|_________________________________________________________________________

	(* Captured Execute *)
	IF EDGEPOS(Execute) THEN
		Internal.CapturedExecute := TRUE;
	ELSIF NOT Execute OR Error THEN
		Internal.CapturedExecute := FALSE;
	END_IF;
	//|_________________________________________________________________________

	//|=========================================================================
	//|					FILLING PROCESS STATE MACHINE
	//|
	//|
	//|=========================================================================
	CASE Internal.Step OF

		//=======================================================
		stepDirCreate_0_Idle: // Idle
			//=======================================================
			Error := FALSE;
			CommandDone := FALSE;
			CommandBusy := FALSE;
			IF Active THEN
				Internal.Step := stepDirCreate_1_WaitCmd;
			END_IF;
			//=======================================================

			//=======================================================
		stepDirCreate_1_WaitCmd: // Wait Cmd
			//=======================================================
			IF (Internal.CapturedExecute) THEN
				CommandBusy := TRUE;
				Internal.Step := stepDirCreate_2_CrateDevLink;
			END_IF;
			//=======================================================

			//=======================================================
		stepDirCreate_2_CrateDevLink:
			//=======================================================
			Internal.FB._DevLink.enable := TRUE;
			Internal.FB._DevLink.pDevice := ADR(Parameters.DeviceName);
			Internal.FB._DevLink.pParam := ADR(Parameters.DirPath);
			Internal.FB._DevLink();
			IF (Internal.FB._DevLink.status = ERR_OK) OR (Internal.FB._DevLink.status = fiERR_DEVICE_ALREADY_EXIST) THEN
				Internal.Step := stepDirCreate_3_CreateDir;
			END_IF;
			//=======================================================

			//=======================================================
		stepDirCreate_3_CreateDir: // Get Dir info
			//=======================================================
			(* Create folder for this component on the user file device *)
			Internal.FB._DirCreate.enable := TRUE;
			Internal.FB._DirCreate.pDevice := ADR(Parameters.DeviceName);
			Internal.FB._DirCreate.pName := ADR('/');
			Internal.FB._DirCreate();
			(* Check if folder already exist and if so disabled the function block call *)
			IF (Internal.FB._DirCreate.status = fiERR_DIR_ALREADY_EXIST) OR (Internal.FB._DirCreate.status = ERR_OK) THEN
				Internal.Step := stepDirCreate_10_Done;
			END_IF
			//=======================================================

			//=======================================================
		stepDirCreate_10_Done: // Done
			//=======================================================
			CommandDone := TRUE;
			IF NOT Execute THEN
				Internal.Step := stepDirCreate_0_Idle;
			END_IF;
			//=======================================================

			//=======================================================
		stepDirCreate_11_Error: // Error
			//=======================================================
			Error := TRUE;
			Internal.FB._DirCreate(enable := FALSE);
			IF ErrorReset THEN
				StatusID := ERR_OK;
				Internal.Step := stepDirCreate_0_Idle;
			END_IF;
		//=======================================================

	END_CASE;
	//|=========================================================================

END_FUNCTION_BLOCK
```

#### FbDirRead.st - Folder içerisindekileri okur.
```iecst
(********************************************************************
 * COPYRIGHT --  B&R Industrial Automation GmbH
 ********************************************************************
 * Library: aLibFile
 * Function Block: FbDirRead
 * Author: kay3a
 * Created: August 27, 2024/4:58 PM
 ********************************************************************
 * Description:  Bu FB parametreden girilen DeviceName de bulunan folder içerisindeki tüm file lati okur.
 ********************************************************************)
FUNCTION_BLOCK FbDirRead

	//|ŻŻŻŻŻŻŻŻŻŻŻŻŻŻŻŻŻŻŻŻŻŻŻŻŻŻŻŻŻŻŻŻŻŻŻŻŻŻŻŻŻŻŻŻŻŻŻŻŻŻŻŻŻŻŻŻŻŻŻŻŻŻŻŻŻŻŻŻŻŻŻŻŻ
	//|               FB ENABLE KONTROLU
	//|_________________________________________________________________________

	(* Enable gelirse FB aktiftir. Gelmiyorsa aktif degildir.  *)
	Active := Enable;

	(* Aktif degilse Step basa gelsin *)
	IF NOT Active THEN
		Internal.Step := stepDirRead_0_Idle;
	END_IF;
	//|_________________________________________________________________________

	//|ŻŻŻŻŻŻŻŻŻŻŻŻŻŻŻŻŻŻŻŻŻŻŻŻŻŻŻŻŻŻŻŻŻŻŻŻŻŻŻŻŻŻŻŻŻŻŻŻŻŻŻŻŻŻŻŻŻŻŻŻŻŻŻŻŻŻŻŻŻŻŻŻŻ
	//|               CHECK FB ERROR
	//|_________________________________________________________________________

	(* Error check *)
	IF (Internal.FB._DirInfo.enable AND Internal.FB._DirInfo.status <> ERR_FUB_BUSY AND Internal.FB._DirInfo.status <> ERR_OK) THEN
		StatusID := Internal.FB._DirInfo.status;
		Internal.Step := stepDirRead_11_Error;

	ELSIF (Internal.FB._DirRead.enable AND Internal.FB._DirRead.status <> ERR_FUB_BUSY AND Internal.FB._DirRead.status <> ERR_OK) THEN
		StatusID := Internal.FB._DirRead.status;
		Internal.Step := stepDirRead_11_Error;
	END_IF;
	//|_________________________________________________________________________

	//|ŻŻŻŻŻŻŻŻŻŻŻŻŻŻŻŻŻŻŻŻŻŻŻŻŻŻŻŻŻŻŻŻŻŻŻŻŻŻŻŻŻŻŻŻŻŻŻŻŻŻŻŻŻŻŻŻŻŻŻŻŻŻŻŻŻŻŻŻŻŻŻŻŻ
	//|               CHECK CMD FB EXECUTE
	//|_________________________________________________________________________

	(* Captured Execute *)
	IF EDGEPOS(Execute) THEN
		Internal.CapturedExecute := TRUE;
	ELSIF NOT Execute OR Error THEN
		Internal.CapturedExecute := FALSE;
	END_IF;
	//|_________________________________________________________________________

	//|=========================================================================
	//|					FILLING PROCESS STATE MACHINE
	//|
	//|
	//|=========================================================================
	CASE Internal.Step OF

		//=======================================================
		stepDirRead_0_Idle: // Idle
			//=======================================================
			Error := FALSE;
			CommandDone := FALSE;
			CommandBusy := FALSE;
			IF Active THEN
				Internal.Step := stepDirRead_1_WaitCmd;
			ELSE
				brsmemset(ADR(ListedFile), 0, SIZEOF(ListedFile));
			END_IF;
			//=======================================================

			//=======================================================
		stepDirRead_1_WaitCmd: // Wait Cmd
			//=======================================================
			IF (Internal.CapturedExecute) THEN
				CommandBusy := TRUE;
				Internal.Step := stepDirRead_2_GetInfo;
			END_IF;
			//=======================================================

			//=======================================================
		stepDirRead_2_GetInfo: // Get Dir info
			//=======================================================
			Internal.FB._DirInfo.enable := TRUE;
			Internal.FB._DirInfo.pDevice := ADR(Parameters.DeviceName);  (* name of the device *)
			Internal.FB._DirInfo.pPath := 0;
			Internal.FB._DirInfo();  (* call the function*)

			IF Internal.FB._DirInfo.status = 0 THEN  (* DirInfo successful *)
				Internal.CountFile := 0;  (* reset Internal.CountFile *)
				brsmemset( ADR(ListedFile), 0, SIZEOF(ListedFile) );  (* clear list*)
				Internal.Step := stepDirRead_3_Read;  (* next step*)
			ELSIF Internal.FB._DirInfo.status = ERR_FUB_BUSY THEN  (* DirInfo not finished -> redo *)
				(* Busy *)
			ELSE  (* Goto internal.status.errorID Step *)
				Internal.Step := stepDirRead_11_Error;
			END_IF
			//=======================================================

			//=======================================================
		stepDirRead_3_Read: // Dir Read
			//=======================================================
			Internal.FB._DirRead.enable := TRUE;
			Internal.FB._DirRead.pDevice := ADR(Parameters.DeviceName);  (* name of the device *)
			Internal.FB._DirRead.pPath := 0;
			Internal.FB._DirRead.option := fiBOTH;  (* read files and folders *)
			Internal.FB._DirRead.entry := Internal.CountFile;
			Internal.FB._DirRead.pData := ADR(Internal.ReadFile);
			Internal.FB._DirRead.data_len := SIZEOF(Internal.ReadFile);
			Internal.FB._DirRead();  (* call the function*)

			IF Internal.FB._DirRead.status = 0 THEN  (* DirRead successful *)
				(* copy found name into string-array *)
				brsstrcpy( ADR(ListedFile[Internal.CountFile]), ADR(Internal.ReadFile.Filename[0]) );
				(* increase Internal.CountFile *)
				Internal.CountFile := Internal.CountFile + 1;
				(* are all files and folders readed out? *)
				IF ( Internal.CountFile < (Internal.FB._DirInfo.dirnum + Internal.FB._DirInfo.filenum) ) THEN
					Internal.Step := stepDirRead_3_Read;  (* read next element *)
				ELSE
					Internal.Step := stepDirRead_10_Done;  (* next step *)
				END_IF
			ELSIF Internal.FB._DirRead.status = ERR_FUB_BUSY THEN  (* DirRead not finished -> redo *)
				(* Busy *)
			ELSE  (* Goto internal.status.errorID Step *)
				Internal.Step := stepDirRead_11_Error;
			END_IF
			//=======================================================

			//=======================================================
		stepDirRead_10_Done: // Done
			//=======================================================
			CommandDone := TRUE;
			IF NOT Execute THEN
				Internal.Step := stepDirRead_0_Idle;
			END_IF;
			//=======================================================

			//=======================================================
		stepDirRead_11_Error: // Error
			//=======================================================
			Error := TRUE;
			Internal.FB._DirInfo(enable := FALSE);
			Internal.FB._DirRead(enable := FALSE);
			IF ErrorReset THEN
				StatusID := ERR_OK;
				Internal.Step := stepDirRead_0_Idle;
			END_IF;
		//=======================================================

	END_CASE;
	//|=========================================================================

END_FUNCTION_BLOCK
```
